gfCNCPoint4[27591] = {X 66.0153, Y 23.5146, Z -6.3333, A 0.000, B 0.000, C 0.000 }
gfCNCPoint4[27592] = {X 71.9863, Y 39.5865, Z -6.3333, A 0.000, B 0.000, C 0.000 }
gfCNCPoint4[27593] = {X 72.3293, Y 40.4492, Z -6.3333, A 0.000, B 0.000, C 0.000 }
gfCNCPoint4[27594] = {X 73.1530, Y 40.9156, Z -6.3333, A 0.000, B 0.000, C 0.000 }
gfCNCPoint4[27595] = {X 73.8471, Y 41.5593, Z -6.3333, A 0.000, B 0.000, C 0.000 }
gfCNCPoint4[27596] = {X 74.3742, Y 42.3456, Z -6.3333, A 0.000, B 0.000, C 0.000 }
gfCNCPoint4[27597] = {X 74.7059, Y 43.2322, Z -6.3333, A 0.000, B 0.000, C 0.000 }
gfCNCPoint4[27598] = {X 74.8243, Y 44.1714, Z -6.3333, A 0.000, B 0.000, C 0.000 }
gfCNCPoint4[27599] = {X 74.8245, Y 45.0000, Z -6.3333, A 0.000, B 0.000, C 0.000 }
gfCNCPoint4[27600] = {X 74.7222, Y 45.9079, Z -6.3333, A 0.000, B 0.000, C 0.000 }
gfCNCPoint4[27601] = {X 74.4204, Y 46.7702, Z -6.3333, A 0.000, B 0.000, C 0.000 }
gfCNCPoint4[27602] = {X 73.9343, Y 47.5438, Z -6.3333, A 0.000, B 0.000, C 0.000 }
gfCNCPoint4[27603] = {X 73.2883, Y 48.1899, Z -6.3333, A 0.000, B 0.000, C 0.000 }
gfCNCPoint4[27604] = {X 72.5147, Y 48.6760, Z -6.3333, A 0.000, B 0.000, C 0.000 }
gfCNCPoint4[27605] = {X 71.6523, Y 48.9777, Z -6.3333, A 0.000, B 0.000, C 0.000 }
gfCNCPoint4[27606] = {X 70.7445, Y 49.0800, Z -6.3333, A 0.000, B 0.000, C 0.000 }
gfCNCPoint4[27607] = {X 64.1851, Y 49.0800, Z -6.3333, A 0.000, B 0.000, C 0.000 }
gfCNCPoint4[27608] = {X 63.2772, Y 48.9777, Z -6.3333, A 0.000, B 0.000, C 0.000 }
gfCNCPoint4[27609] = {X 62.4149, Y 48.6760, Z -6.3333, A 0.000, B 0.000, C 0.000 }
gfCNCPoint4[27610] = {X 61.6413, Y 48.1899, Z -6.3333, A 0.000, B 0.000, C 0.000 }
gfCNCPoint4[27611] = {X 60.9953, Y 47.5438, Z -6.3333, A 0.000, B 0.000, C 0.000 }
gfCNCPoint4[27612] = {X 60.5092, Y 46.7702, Z -6.3333, A 0.000, B 0.000, C 0.000 }
gfCNCPoint4[27613] = {X 60.2074, Y 45.9079, Z -6.3333, A 0.000, B 0.000, C 0.000 }
gfCNCPoint4[27614] = {X 60.1051, Y 45.0000, Z -6.3333, A 0.000, B 0.000, C 0.000 }
gfCNCPoint4[27615] = {X 60.1051, Y 44.2086, Z -6.3333, A 0.000, B 0.000, C 0.000 }
gfCNCPoint4[27616] = {X 60.1952, Y 43.3581, Z -6.3333, A 0.000, B 0.000, C 0.000 }
gfCNCPoint4[27617] = {X 60.4606, Y 42.5451, Z -6.3333, A 0.000, B 0.000, C 0.000 }
gfCNCPoint4[27618] = {X 60.8897, Y 41.8052, Z -6.3333, A 0.000, B 0.000, C 0.000 }
gfCNCPoint4[27619] = {X 60.1744, Y 39.8492, Z -6.3333, A 0.000, B 0.000, C 0.000 }
gfCNCPoint4[27620] = {X 51.9112, Y 39.8492, Z -6.3333, A 0.000, B 0.000, C 0.000 }
gfCNCPoint4[27621] = {X 51.0699, Y 42.1094, Z -6.3333, A 0.000, B 0.000, C 0.000 }
gfCNCPoint4[27622] = {X 51.1301, Y 42.2106, Z -6.3333, A 0.000, B 0.000, C 0.000 }
gfCNCPoint4[27623] = {X 51.4138, Y 42.8326, Z -6.3333, A 0.000, B 0.000, C 0.000 }
gfCNCPoint4[27624] = {X 51.5897, Y 43.4933, Z -6.3333, A 0.000, B 0.000, C 0.000 }
gfCNCPoint4[27625] = {X 51.6528, Y 44.1740, Z -6.3333, A 0.000, B 0.000, C 0.000 }
gfCNCPoint4[27626] = {X 51.6529, Y 45.0000, Z -6.3333, A 0.000, B 0.000, C 0.000 }
gfCNCPoint4[27627] = {X 51.5506, Y 45.9079, Z -6.3333, A 0.000, B 0.000, C 0.000 }
gfCNCPoint4[27628] = {X 51.2489, Y 46.7702, Z -6.3333, A 0.000, B 0.000, C 0.000 }
gfCNCPoint4[27629] = {X 50.7628, Y 47.5438, Z -6.3333, A 0.000, B 0.000, C 0.000 }
gfCNCPoint4[27630] = {X 50.1168, Y 48.1899, Z -6.3333, A 0.000, B 0.000, C 0.000 }
gfCNCPoint4[27631] = {X 49.3432, Y 48.6760, Z -6.3333, A 0.000, B 0.000, C 0.000 }
gfCNCPoint4[27632] = {X 48.4808, Y 48.9777, Z -6.3333, A 0.000, B 0.000, C 0.000 }
gfCNCPoint4[27633] = {X 47.5729, Y 49.0800, Z -6.3333, A 0.000, B 0.000, C 0.000 }
gfCNCPoint4[27634] = {X 40.6393, Y 49.0800, Z -6.3333, A 0.000, B 0.000, C 0.000 }
gfCNCPoint4[27635] = {X 39.7314, Y 48.9777, Z -6.3333, A 0.000, B 0.000, C 0.000 }
gfCNCPoint4[27636] = {X 38.8691, Y 48.6760, Z -6.3333, A 0.000, B 0.000, C 0.000 }
gfCNCPoint4[27637] = {X 38.0955, Y 48.1899, Z -6.3333, A 0.000, B 0.000, C 0.000 }
gfCNCPoint4[27638] = {X 37.4494, Y 47.5438, Z -6.3333, A 0.000, B 0.000, C 0.000 }
gfCNCPoint4[27639] = {X 36.9633, Y 46.7702, Z -6.3333, A 0.000, B 0.000, C 0.000 }
gfCNCPoint4[27640] = {X 36.6616, Y 45.9079, Z -6.3333, A 0.000, B 0.000, C 0.000 }
gfCNCPoint4[27641] = {X 36.5593, Y 45.0000, Z -6.3333, A 0.000, B 0.000, C 0.000 }
gfCNCPoint4[27642] = {X 36.5593, Y 44.2086, Z -6.3333, A 0.000, B 0.000, C 0.000 }
gfCNCPoint4[27643] = {X 36.6734, Y 43.2505, Z -6.3333, A 0.000, B 0.000, C 0.000 }
gfCNCPoint4[27644] = {X 37.0093, Y 42.3461, Z -6.3333, A 0.000, B 0.000, C 0.000 }
gfCNCPoint4[27645] = {X 37.5482, Y 41.5458, Z -6.3333, A 0.000, B 0.000, C 0.000 }
gfCNCPoint4[27646] = {X 38.2600, Y 40.8944, Z -6.3333, A 0.000, B 0.000, C 0.000 }
gfCNCPoint4[27647] = {X 39.1048, Y 40.4284, Z -6.3333, A 0.000, B 0.000, C 0.000 }
gfCNCPoint4[27648] = {X 39.1153, Y 40.4182, Z -6.3333, A 0.000, B 0.000, C 0.000 }
gfCNCPoint4[27649] = {X 39.1252, Y 40.3961, Z -6.3333, A 0.000, B 0.000, C 0.000 }
gfCNCPoint4[27650] = {X 39.7337, Y 38.9641, Z -6.3333, A 0.000, B 0.000, C 0.000 }
gfCNCPoint4[27651] = {X 40.2895, Y 37.5107, Z -6.3333, A 0.000, B 0.000, C 0.000 }
gfCNCPoint4[27652] = {X 43.8728, Y 27.8910, Z -6.3333, A 0.000, B 0.000, C 0.000 }
gfCNCPoint4[27653] = {X 40.1244, Y 26.4948, Z -6.3333, A 0.000, B 0.000, C 0.000 }
gfCNCPoint4[27654] = {X 43.9477, Y 27.9190, Z -6.3333, A 0.000, B 0.000, C 0.000 }
gfCNCPoint4[27655] = {X 48.6479, Y 15.3010, Z -6.3333, A 0.000, B 0.000, C 0.000 }
gfCNCPoint4[27656] = {X 48.2407, Y 14.5838, Z -6.3333, A 0.000, B 0.000, C 0.000 }
gfCNCPoint4[27657] = {X 47.9892, Y 13.7983, Z -6.3333, A 0.000, B 0.000, C 0.000 }
gfCNCPoint4[27658] = {X 47.9042, Y 12.9780, Z -6.3333, A 0.000, B 0.000, C 0.000 }
gfCNCPoint4[27659] = {X 47.9042, Y 12.1868, Z -6.3333, A 0.000, B 0.000, C 0.000 }
gfCNCPoint4[27660] = {X 48.0045, Y 11.2967, Z -6.3333, A 0.000, B 0.000, C 0.000 }
gfCNCPoint4[27661] = {X 48.3003, Y 10.4513, Z -6.3333, A 0.000, B 0.000, C 0.000 }
gfCNCPoint4[27662] = {X 48.7769, Y 9.6929, Z -6.3333, A 0.000, B 0.000, C 0.000 }
gfCNCPoint4[27663] = {X 49.4103, Y 9.0595, Z -6.3333, A 0.000, B 0.000, C 0.000 }
gfCNCPoint4[27664] = {X 50.1687, Y 8.5829, Z -6.3333, A 0.000, B 0.000, C 0.000 }
gfCNCPoint4[27665] = {X 51.0141, Y 8.2871, Z -6.3333, A 0.000, B 0.000, C 0.000 }
gfCNCPoint4[27666] = {X 51.9042, Y 8.1868, Z -6.3333, A 0.000, B 0.000, C 0.000 }
gfCNCPoint4[27667] = {X 59.6221, Y 8.1868, Z -6.3333, A 0.000, B 0.000, C 0.000 }
gfCNCPoint4[27668] = {X 60.5122, Y 8.2871, Z -6.3333, A 0.000, B 0.000, C 0.000 }
gfCNCPoint4[27669] = {X 61.3577, Y 8.5829, Z -6.3333, A 0.000, B 0.000, C 0.000 }
gfCNCPoint4[27670] = {X 62.1161, Y 9.0595, Z -6.3333, A 0.000, B 0.000, C 0.000 }
gfCNCPoint4[27671] = {X 62.7495, Y 9.6929, Z -6.3333, A 0.000, B 0.000, C 0.000 }
gfCNCPoint4[27672] = {X 63.2260, Y 10.4513, Z -6.3333, A 0.000, B 0.000, C 0.000 }
gfCNCPoint4[27673] = {X 63.5218, Y 11.2967, Z -6.3333, A 0.000, B 0.000, C 0.000 }
gfCNCPoint4[27674] = {X 63.6221, Y 12.1868, Z -6.3333, A 0.000, B 0.000, C 0.000 }
gfCNCPoint4[27675] = {X 63.6219, Y 13.0192, Z -6.3333, A 0.000, B 0.000, C 0.000 }
gfCNCPoint4[27676] = {X 63.5278, Y 13.8417, Z -6.3333, A 0.000, B 0.000, C 0.000 }
gfCNCPoint4[27677] = {X 63.2663, Y 14.6272, Z -6.3333, A 0.000, B 0.000, C 0.000 }
gfCNCPoint4[27678] = {X 62.8488, Y 15.3420, Z -6.3333, A 0.000, B 0.000, C 0.000 }
gfCNCPoint4[27679] = {X 63.1271, Y 16.0764, Z -6.3333, A 0.000, B 0.000, C 0.000 }
gfCNCPoint4[27680] = {X 65.9404, Y 23.5426, Z -6.3333, A 0.000, B 0.000, C 0.000 }
gfCNCPoint4[27681] = {X 71.9117, Y 39.6152, Z -6.3333, A 0.000, B 0.000, C 0.000 }
gfCNCPoint4[27682] = {X 72.2608, Y 40.4935, Z -6.3333, A 0.000, B 0.000, C 0.000 }
gfCNCPoint4[27683] = {X 72.2699, Y 40.5075, Z -6.3333, A 0.000, B 0.000, C 0.000 }
gfCNCPoint4[27684] = {X 72.2838, Y 40.5168, Z -6.3333, A 0.000, B 0.000, C 0.000 }
gfCNCPoint4[27685] = {X 72.3479, Y 40.5442, Z -6.3333, A 0.000, B 0.000, C 0.000 }
gfCNCPoint4[27686] = {X 72.4115, Y 40.5727, Z -6.3333, A 0.000, B 0.000, C 0.000 }
gfCNCPoint4[27687] = {X 73.1908, Y 41.0441, Z -6.3333, A 0.000, B 0.000, C 0.000 }
gfCNCPoint4[27688] = {X 73.8433, Y 41.6795, Z -6.3333, A 0.000, B 0.000, C 0.000 }
gfCNCPoint4[27689] = {X 74.3351, Y 42.4461, Z -6.3333, A 0.000, B 0.000, C 0.000 }
gfCNCPoint4[27690] = {X 74.6408, Y 43.3040, Z -6.3333, A 0.000, B 0.000, C 0.000 }
gfCNCPoint4[27691] = {X 74.7445, Y 44.2089, Z -6.3333, A 0.000, B 0.000, C 0.000 }
gfCNCPoint4[27692] = {X 74.7445, Y 45.0000, Z -6.3333, A 0.000, B 0.000, C 0.000 }
gfCNCPoint4[27693] = {X 74.6442, Y 45.8901, Z -6.3333, A 0.000, B 0.000, C 0.000 }
gfCNCPoint4[27694] = {X 74.3483, Y 46.7355, Z -6.3333, A 0.000, B 0.000, C 0.000 }
gfCNCPoint4[27695] = {X 73.8718, Y 47.4940, Z -6.3333, A 0.000, B 0.000, C 0.000 }
gfCNCPoint4[27696] = {X 73.2384, Y 48.1273, Z -6.3333, A 0.000, B 0.000, C 0.000 }
gfCNCPoint4[27697] = {X 72.4800, Y 48.6039, Z -6.3333, A 0.000, B 0.000, C 0.000 }
gfCNCPoint4[27698] = {X 71.6345, Y 48.8997, Z -6.3333, A 0.000, B 0.000, C 0.000 }
gfCNCPoint4[27699] = {X 70.7445, Y 49.0000, Z -6.3333, A 0.000, B 0.000, C 0.000 }
gfCNCPoint4[27700] = {X 64.1851, Y 49.0000, Z -6.3333, A 0.000, B 0.000, C 0.000 }
gfCNCPoint4[27701] = {X 63.2951, Y 48.8997, Z -6.3333, A 0.000, B 0.000, C 0.000 }
gfCNCPoint4[27702] = {X 62.4496, Y 48.6039, Z -6.3333, A 0.000, B 0.000, C 0.000 }
gfCNCPoint4[27703] = {X 61.6912, Y 48.1273, Z -6.3333, A 0.000, B 0.000, C 0.000 }
gfCNCPoint4[27704] = {X 61.0578, Y 47.4940, Z -6.3333, A 0.000, B 0.000, C 0.000 }
gfCNCPoint4[27705] = {X 60.5813, Y 46.7355, Z -6.3333, A 0.000, B 0.000, C 0.000 }
gfCNCPoint4[27706] = {X 60.2854, Y 45.8901, Z -6.3333, A 0.000, B 0.000, C 0.000 }
gfCNCPoint4[27707] = {X 60.1851, Y 45.0000, Z -6.3333, A 0.000, B 0.000, C 0.000 }
gfCNCPoint4[27708] = {X 60.1855, Y 44.1538, Z -6.3333, A 0.000, B 0.000, C 0.000 }
gfCNCPoint4[27709] = {X 60.2746, Y 43.3674, Z -6.3333, A 0.000, B 0.000, C 0.000 }
gfCNCPoint4[27710] = {X 60.5168, Y 42.6140, Z -6.3333, A 0.000, B 0.000, C 0.000 }
gfCNCPoint4[27711] = {X 60.9025, Y 41.9231, Z -6.3333, A 0.000, B 0.000, C 0.000 }
gfCNCPoint4[27712] = {X 60.9795, Y 41.8179, Z -6.3333, A 0.000, B 0.000, C 0.000 }
gfCNCPoint4[27713] = {X 60.2304, Y 39.7692, Z -6.3333, A 0.000, B 0.000, C 0.000 }
gfCNCPoint4[27714] = {X 51.8428, Y 39.7692, Z -6.3333, A 0.000, B 0.000, C 0.000 }
gfCNCPoint4[27715] = {X 51.8428, Y 39.8035, Z -6.3333, A 0.000, B 0.000, C 0.000 }
gfCNCPoint4[27716] = {X 50.9816, Y 42.1174, Z -6.3333, A 0.000, B 0.000, C 0.000 }
gfCNCPoint4[27717] = {X 51.0729, Y 42.2722, Z -6.3333, A 0.000, B 0.000, C 0.000 }
gfCNCPoint4[27718] = {X 51.3480, Y 42.8865, Z -6.3333, A 0.000, B 0.000, C 0.000 }
gfCNCPoint4[27719] = {X 51.5163, Y 43.5382, Z -6.3333, A 0.000, B 0.000, C 0.000 }
gfCNCPoint4[27720] = {X 51.5729, Y 44.2089, Z -6.3333, A 0.000, B 0.000, C 0.000 }
gfCNCPoint4[27721] = {X 51.5729, Y 45.0000, Z -6.3333, A 0.000, B 0.000, C 0.000 }
gfCNCPoint4[27722] = {X 51.4726, Y 45.8901, Z -6.3333, A 0.000, B 0.000, C 0.000 }
gfCNCPoint4[27723] = {X 51.1768, Y 46.7355, Z -6.3333, A 0.000, B 0.000, C 0.000 }
gfCNCPoint4[27724] = {X 50.7003, Y 47.4940, Z -6.3333, A 0.000, B 0.000, C 0.000 }
gfCNCPoint4[27725] = {X 50.0669, Y 48.1273, Z -6.3333, A 0.000, B 0.000, C 0.000 }
gfCNCPoint4[27726] = {X 49.3085, Y 48.6039, Z -6.3333, A 0.000, B 0.000, C 0.000 }
gfCNCPoint4[27727] = {X 48.4630, Y 48.8997, Z -6.3333, A 0.000, B 0.000, C 0.000 }
gfCNCPoint4[27728] = {X 47.5729, Y 49.0000, Z -6.3333, A 0.000, B 0.000, C 0.000 }
gfCNCPoint4[27729] = {X 40.6393, Y 49.0000, Z -6.3333, A 0.000, B 0.000, C 0.000 }
gfCNCPoint4[27730] = {X 39.7492, Y 48.8997, Z -6.3333, A 0.000, B 0.000, C 0.000 }
gfCNCPoint4[27731] = {X 38.9038, Y 48.6039, Z -6.3333, A 0.000, B 0.000, C 0.000 }
gfCNCPoint4[27732] = {X 38.1453, Y 48.1273, Z -6.3333, A 0.000, B 0.000, C 0.000 }
gfCNCPoint4[27733] = {X 37.5120, Y 47.4940, Z -6.3333, A 0.000, B 0.000, C 0.000 }
gfCNCPoint4[27734] = {X 37.0354, Y 46.7355, Z -6.3333, A 0.000, B 0.000, C 0.000 }
gfCNCPoint4[27735] = {X 36.7396, Y 45.8901, Z -6.3333, A 0.000, B 0.000, C 0.000 }
gfCNCPoint4[27736] = {X 36.6393, Y 45.0000, Z -6.3333, A 0.000, B 0.000, C 0.000 }
gfCNCPoint4[27737] = {X 36.6397, Y 44.1538, Z -6.3333, A 0.000, B 0.000, C 0.000 }
gfCNCPoint4[27738] = {X 36.7563, Y 43.2484, Z -6.3333, A 0.000, B 0.000, C 0.000 }
gfCNCPoint4[27739] = {X 37.0752, Y 42.3931, Z -6.3333, A 0.000, B 0.000, C 0.000 }
gfCNCPoint4[27740] = {X 37.5796, Y 41.6323, Z -6.3333, A 0.000, B 0.000, C 0.000 }
gfCNCPoint4[27741] = {X 38.2434, Y 41.0057, Z -6.3333, A 0.000, B 0.000, C 0.000 }
gfCNCPoint4[27742] = {X 39.0320, Y 40.5459, Z -6.3333, A 0.000, B 0.000, C 0.000 }
gfCNCPoint4[27743] = {X 39.0833, Y 40.5238, Z -6.3333, A 0.000, B 0.000, C 0.000 }
gfCNCPoint4[27744] = {X 39.1349, Y 40.5025, Z -6.3333, A 0.000, B 0.000, C 0.000 }
gfCNCPoint4[27745] = {X 39.1666, Y 40.4818, Z -6.3333, A 0.000, B 0.000, C 0.000 }
gfCNCPoint4[27746] = {X 39.1883, Y 40.4509, Z -6.3333, A 0.000, B 0.000, C 0.000 }
gfCNCPoint4[27747] = {X 39.2126, Y 40.3964, Z -6.3333, A 0.000, B 0.000, C 0.000 }
gfCNCPoint4[27748] = {X 39.2369, Y 40.3420, Z -6.3333, A 0.000, B 0.000, C 0.000 }
gfCNCPoint4[27749] = {X 39.8256, Y 38.9501, Z -6.3333, A 0.000, B 0.000, C 0.000 }
gfCNCPoint4[27750] = {X 40.3646, Y 37.5383, Z -6.3333, A 0.000, B 0.000, C 0.000 }
gfCNCPoint4[27751] = {X 43.9477, Y 27.9190, Z -6.3333, A 0.000, B 0.000, C 0.000 }
gfCNCPoint4[27752] = {X 40.1244, Y 26.4948, Z -6.3333, A 0.000, B 0.000, C 0.000 }
gfCNCPoint4[27753] = {X 40.1244, Y 26.4948, Z -3.3333, A 0.000, B 0.000, C 0.000 }
gfCNCPoint4[27754] = {X 40.1244, Y 26.4948, Z 11.0000, A 0.000, B 0.000, C 0.000 }
gfCNCPoint4[27755] = {X 79.0220, Y 28.5912, Z 11.0000, A 0.000, B 0.000, C 0.000 }
gfCNCPoint4[27756] = {X 79.0220, Y 28.5912, Z -3.3333, A 0.000, B 0.000, C 0.000 }
gfCNCPoint4[27757] = {X 79.0220, Y 28.5912, Z -6.3333, A 0.000, B 0.000, C 0.000 }
gfCNCPoint4[27758] = {X 83.1020, Y 28.5912, Z -6.3333, A 0.000, B 0.000, C 0.000 }
gfCNCPoint4[27759] = {X 83.1019, Y 16.2736, Z -6.3333, A 0.000, B 0.000, C 0.000 }
gfCNCPoint4[27760] = {X 82.4637, Y 15.6025, Z -6.3333, A 0.000, B 0.000, C 0.000 }
gfCNCPoint4[27761] = {X 81.9831, Y 14.8108, Z -6.3333, A 0.000, B 0.000, C 0.000 }
gfCNCPoint4[27762] = {X 81.6824, Y 13.9349, Z -6.3333, A 0.000, B 0.000, C 0.000 }
gfCNCPoint4[27763] = {X 81.5752, Y 13.0150, Z -6.3333, A 0.000, B 0.000, C 0.000 }
gfCNCPoint4[27764] = {X 81.5751, Y 12.1868, Z -6.3333, A 0.000, B 0.000, C 0.000 }
gfCNCPoint4[27765] = {X 81.6834, Y 11.2255, Z -6.3333, A 0.000, B 0.000, C 0.000 }
gfCNCPoint4[27766] = {X 82.0029, Y 10.3125, Z -6.3333, A 0.000, B 0.000, C 0.000 }
gfCNCPoint4[27767] = {X 82.5176, Y 9.4933, Z -6.3333, A 0.000, B 0.000, C 0.000 }
gfCNCPoint4[27768] = {X 83.2016, Y 8.8093, Z -6.3333, A 0.000, B 0.000, C 0.000 }
gfCNCPoint4[27769] = {X 84.0207, Y 8.2946, Z -6.3333, A 0.000, B 0.000, C 0.000 }
gfCNCPoint4[27770] = {X 84.9338, Y 7.9751, Z -6.3333, A 0.000, B 0.000, C 0.000 }
gfCNCPoint4[27771] = {X 85.8951, Y 7.8668, Z -6.3333, A 0.000, B 0.000, C 0.000 }
gfCNCPoint4[27772] = {X 94.0497, Y 7.8668, Z -6.3333, A 0.000, B 0.000, C 0.000 }
gfCNCPoint4[27773] = {X 95.0110, Y 7.9751, Z -6.3333, A 0.000, B 0.000, C 0.000 }
gfCNCPoint4[27774] = {X 95.9240, Y 8.2946, Z -6.3333, A 0.000, B 0.000, C 0.000 }
gfCNCPoint4[27775] = {X 96.7431, Y 8.8093, Z -6.3333, A 0.000, B 0.000, C 0.000 }
gfCNCPoint4[27776] = {X 97.4272, Y 9.4933, Z -6.3333, A 0.000, B 0.000, C 0.000 }
gfCNCPoint4[27777] = {X 97.9419, Y 10.3124, Z -6.3333, A 0.000, B 0.000, C 0.000 }
gfCNCPoint4[27778] = {X 98.2614, Y 11.2255, Z -6.3333, A 0.000, B 0.000, C 0.000 }
gfCNCPoint4[27779] = {X 98.3697, Y 12.1868, Z -6.3333, A 0.000, B 0.000, C 0.000 }
gfCNCPoint4[27780] = {X 98.3697, Y 12.9782, Z -6.3333, A 0.000, B 0.000, C 0.000 }
gfCNCPoint4[27781] = {X 98.2967, Y 13.7678, Z -6.3333, A 0.000, B 0.000, C 0.000 }
gfCNCPoint4[27782] = {X 98.0807, Y 14.5307, Z -6.3333, A 0.000, B 0.000, C 0.000 }
gfCNCPoint4[27783] = {X 97.7289, Y 15.2414, Z -6.3333, A 0.000, B 0.000, C 0.000 }
gfCNCPoint4[27784] = {X 101.8758, Y 25.5228, Z -6.3333, A 0.000, B 0.000, C 0.000 }
gfCNCPoint4[27785] = {X 106.0162, Y 15.2210, Z -6.3333, A 0.000, B 0.000, C 0.000 }
gfCNCPoint4[27786] = {X 105.6760, Y 14.5282, Z -6.3333, A 0.000, B 0.000, C 0.000 }
gfCNCPoint4[27787] = {X 105.4645, Y 13.7860, Z -6.3333, A 0.000, B 0.000, C 0.000 }
gfCNCPoint4[27788] = {X 105.3885, Y 13.0179, Z -6.3333, A 0.000, B 0.000, C 0.000 }
gfCNCPoint4[27789] = {X 105.3883, Y 12.1868, Z -6.3333, A 0.000, B 0.000, C 0.000 }
gfCNCPoint4[27790] = {X 105.4966, Y 11.2255, Z -6.3333, A 0.000, B 0.000, C 0.000 }
gfCNCPoint4[27791] = {X 105.8161, Y 10.3124, Z -6.3333, A 0.000, B 0.000, C 0.000 }
gfCNCPoint4[27792] = {X 106.3308, Y 9.4933, Z -6.3333, A 0.000, B 0.000, C 0.000 }
gfCNCPoint4[27793] = {X 107.0148, Y 8.8093, Z -6.3333, A 0.000, B 0.000, C 0.000 }
gfCNCPoint4[27794] = {X 107.8339, Y 8.2946, Z -6.3333, A 0.000, B 0.000, C 0.000 }
gfCNCPoint4[27795] = {X 108.7470, Y 7.9751, Z -6.3333, A 0.000, B 0.000, C 0.000 }
gfCNCPoint4[27796] = {X 109.7083, Y 7.8668, Z -6.3333, A 0.000, B 0.000, C 0.000 }
gfCNCPoint4[27797] = {X 117.7916, Y 7.8668, Z -6.3333, A 0.000, B 0.000, C 0.000 }
gfCNCPoint4[27798] = {X 118.7529, Y 7.9751, Z -6.3333, A 0.000, B 0.000, C 0.000 }
gfCNCPoint4[27799] = {X 119.6660, Y 8.2946, Z -6.3333, A 0.000, B 0.000, C 0.000 }
gfCNCPoint4[27800] = {X 120.4851, Y 8.8093, Z -6.3333, A 0.000, B 0.000, C 0.000 }
gfCNCPoint4[27801] = {X 121.1691, Y 9.4933, Z -6.3333, A 0.000, B 0.000, C 0.000 }
gfCNCPoint4[27802] = {X 121.6838, Y 10.3124, Z -6.3333, A 0.000, B 0.000, C 0.000 }
gfCNCPoint4[27803] = {X 122.0033, Y 11.2255, Z -6.3333, A 0.000, B 0.000, C 0.000 }
gfCNCPoint4[27804] = {X 122.1116, Y 12.1868, Z -6.3333, A 0.000, B 0.000, C 0.000 }
gfCNCPoint4[27805] = {X 122.1116, Y 12.9782, Z -6.3333, A 0.000, B 0.000, C 0.000 }
gfCNCPoint4[27806] = {X 122.0103, Y 13.9078, Z -6.3333, A 0.000, B 0.000, C 0.000 }
gfCNCPoint4[27807] = {X 121.7114, Y 14.7939, Z -6.3333, A 0.000, B 0.000, C 0.000 }
gfCNCPoint4[27808] = {X 121.2288, Y 15.5949, Z -6.3333, A 0.000, B 0.000, C 0.000 }
gfCNCPoint4[27809] = {X 120.5851, Y 16.2732, Z -6.3333, A 0.000, B 0.000, C 0.000 }
gfCNCPoint4[27810] = {X 120.5847, Y 40.9145, Z -6.3333, A 0.000, B 0.000, C 0.000 }
gfCNCPoint4[27811] = {X 120.6226, Y 40.9457, Z -6.3333, A 0.000, B 0.000, C 0.000 }
gfCNCPoint4[27812] = {X 121.2458, Y 41.6145, Z -6.3333, A 0.000, B 0.000, C 0.000 }
gfCNCPoint4[27813] = {X 121.7144, Y 42.3993, Z -6.3333, A 0.000, B 0.000, C 0.000 }
gfCNCPoint4[27814] = {X 122.0073, Y 43.2652, Z -6.3333, A 0.000, B 0.000, C 0.000 }
gfCNCPoint4[27815] = {X 122.1114, Y 44.1734, Z -6.3333, A 0.000, B 0.000, C 0.000 }
gfCNCPoint4[27816] = {X 122.1116, Y 45.0000, Z -6.3333, A 0.000, B 0.000, C 0.000 }
gfCNCPoint4[27817] = {X 122.0033, Y 45.9613, Z -6.3333, A 0.000, B 0.000, C 0.000 }
gfCNCPoint4[27818] = {X 121.6838, Y 46.8744, Z -6.3333, A 0.000, B 0.000, C 0.000 }
gfCNCPoint4[27819] = {X 121.1691, Y 47.6935, Z -6.3333, A 0.000, B 0.000, C 0.000 }
gfCNCPoint4[27820] = {X 120.4851, Y 48.3775, Z -6.3333, A 0.000, B 0.000, C 0.000 }
gfCNCPoint4[27821] = {X 119.6660, Y 48.8922, Z -6.3333, A 0.000, B 0.000, C 0.000 }
gfCNCPoint4[27822] = {X 118.7529, Y 49.2117, Z -6.3333, A 0.000, B 0.000, C 0.000 }
gfCNCPoint4[27823] = {X 117.7916, Y 49.3200, Z -6.3333, A 0.000, B 0.000, C 0.000 }
gfCNCPoint4[27824] = {X 111.9185, Y 49.3200, Z -6.3333, A 0.000, B 0.000, C 0.000 }
gfCNCPoint4[27825] = {X 110.9619, Y 49.2128, Z -6.3333, A 0.000, B 0.000, C 0.000 }
gfCNCPoint4[27826] = {X 110.0529, Y 48.8964, Z -6.3333, A 0.000, B 0.000, C 0.000 }
gfCNCPoint4[27827] = {X 109.2365, Y 48.3866, Z -6.3333, A 0.000, B 0.000, C 0.000 }
gfCNCPoint4[27828] = {X 108.5532, Y 47.7087, Z -6.3333, A 0.000, B 0.000, C 0.000 }
gfCNCPoint4[27829] = {X 108.0369, Y 46.8963, Z -6.3333, A 0.000, B 0.000, C 0.000 }
gfCNCPoint4[27830] = {X 107.7134, Y 45.9898, Z -6.3333, A 0.000, B 0.000, C 0.000 }
gfCNCPoint4[27831] = {X 107.5986, Y 45.0341, Z -6.3333, A 0.000, B 0.000, C 0.000 }
gfCNCPoint4[27832] = {X 107.5985, Y 44.1789, Z -6.3333, A 0.000, B 0.000, C 0.000 }
gfCNCPoint4[27833] = {X 107.6340, Y 43.6366, Z -6.3333, A 0.000, B 0.000, C 0.000 }
gfCNCPoint4[27834] = {X 107.7400, Y 43.1035, Z -6.3333, A 0.000, B 0.000, C 0.000 }
gfCNCPoint4[27835] = {X 107.9081, Y 42.6047, Z -6.3333, A 0.000, B 0.000, C 0.000 }
gfCNCPoint4[27836] = {X 108.1379, Y 42.1311, Z -6.3333, A 0.000, B 0.000, C 0.000 }
gfCNCPoint4[27837] = {X 108.5875, Y 41.4624, Z -6.3333, A 0.000, B 0.000, C 0.000 }
gfCNCPoint4[27838] = {X 109.1253, Y 40.8623, Z -6.3333, A 0.000, B 0.000, C 0.000 }
gfCNCPoint4[27839] = {X 109.1252, Y 39.2978, Z -6.3333, A 0.000, B 0.000, C 0.000 }
gfCNCPoint4[27840] = {X 106.1118, Y 46.6615, Z -6.3333, A 0.000, B 0.000, C 0.000 }
gfCNCPoint4[27841] = {X 105.7417, Y 47.3611, Z -6.3333, A 0.000, B 0.000, C 0.000 }
gfCNCPoint4[27842] = {X 105.2502, Y 47.9815, Z -6.3333, A 0.000, B 0.000, C 0.000 }
gfCNCPoint4[27843] = {X 104.6538, Y 48.5018, Z -6.3333, A 0.000, B 0.000, C 0.000 }
gfCNCPoint4[27844] = {X 103.9724, Y 48.9046, Z -6.3333, A 0.000, B 0.000, C 0.000 }
gfCNCPoint4[27845] = {X 103.0287, Y 49.2242, Z -6.3333, A 0.000, B 0.000, C 0.000 }
gfCNCPoint4[27846] = {X 102.0368, Y 49.3191, Z -6.3333, A 0.000, B 0.000, C 0.000 }
gfCNCPoint4[27847] = {X 101.0496, Y 49.1842, Z -6.3333, A 0.000, B 0.000, C 0.000 }
gfCNCPoint4[27848] = {X 100.1195, Y 48.8268, Z -6.3333, A 0.000, B 0.000, C 0.000 }
gfCNCPoint4[27849] = {X 99.2961, Y 48.2657, Z -6.3333, A 0.000, B 0.000, C 0.000 }
gfCNCPoint4[27850] = {X 98.6231, Y 47.5309, Z -6.3333, A 0.000, B 0.000, C 0.000 }
gfCNCPoint4[27851] = {X 98.1363, Y 46.6615, Z -6.3333, A 0.000, B 0.000, C 0.000 }
gfCNCPoint4[27852] = {X 95.1317, Y 39.3133, Z -6.3333, A 0.000, B 0.000, C 0.000 }
gfCNCPoint4[27853] = {X 95.1317, Y 40.9048, Z -6.3333, A 0.000, B 0.000, C 0.000 }
gfCNCPoint4[27854] = {X 95.6575, Y 41.4431, Z -6.3333, A 0.000, B 0.000, C 0.000 }
gfCNCPoint4[27855] = {X 96.0839, Y 42.0632, Z -6.3333, A 0.000, B 0.000, C 0.000 }
gfCNCPoint4[27856] = {X 96.3313, Y 42.5720, Z -6.3333, A 0.000, B 0.000, C 0.000 }
gfCNCPoint4[27857] = {X 96.5113, Y 43.1084, Z -6.3333, A 0.000, B 0.000, C 0.000 }
gfCNCPoint4[27858] = {X 96.6196, Y 43.6529, Z -6.3333, A 0.000, B 0.000, C 0.000 }
gfCNCPoint4[27859] = {X 96.6585, Y 44.2066, Z -6.3333, A 0.000, B 0.000, C 0.000 }
gfCNCPoint4[27860] = {X 96.6583, Y 45.0415, Z -6.3333, A 0.000, B 0.000, C 0.000 }
gfCNCPoint4[27861] = {X 96.5422, Y 45.9960, Z -6.3333, A 0.000, B 0.000, C 0.000 }
gfCNCPoint4[27862] = {X 96.2178, Y 46.9011, Z -6.3333, A 0.000, B 0.000, C 0.000 }
gfCNCPoint4[27863] = {X 95.7012, Y 47.7120, Z -6.3333, A 0.000, B 0.000, C 0.000 }
gfCNCPoint4[27864] = {X 95.0181, Y 48.3886, Z -6.3333, A 0.000, B 0.000, C 0.000 }
gfCNCPoint4[27865] = {X 94.2022, Y 48.8973, Z -6.3333, A 0.000, B 0.000, C 0.000 }
gfCNCPoint4[27866] = {X 93.2940, Y 49.2130, Z -6.3333, A 0.000, B 0.000, C 0.000 }
gfCNCPoint4[27867] = {X 92.3385, Y 49.3200, Z -6.3333, A 0.000, B 0.000, C 0.000 }
gfCNCPoint4[27868] = {X 85.8951, Y 49.3200, Z -6.3333, A 0.000, B 0.000, C 0.000 }
gfCNCPoint4[27869] = {X 84.9387, Y 49.2128, Z -6.3333, A 0.000, B 0.000, C 0.000 }
gfCNCPoint4[27870] = {X 84.0297, Y 48.8965, Z -6.3333, A 0.000, B 0.000, C 0.000 }
gfCNCPoint4[27871] = {X 83.2134, Y 48.3869, Z -6.3333, A 0.000, B 0.000, C 0.000 }
gfCNCPoint4[27872] = {X 82.5301, Y 47.7091, Z -6.3333, A 0.000, B 0.000, C 0.000 }
gfCNCPoint4[27873] = {X 82.0138, Y 46.8970, Z -6.3333, A 0.000, B 0.000, C 0.000 }
gfCNCPoint4[27874] = {X 81.6902, Y 45.9906, Z -6.3333, A 0.000, B 0.000, C 0.000 }
gfCNCPoint4[27875] = {X 81.5752, Y 45.0351, Z -6.3333, A 0.000, B 0.000, C 0.000 }
gfCNCPoint4[27876] = {X 81.5751, Y 44.2072, Z -6.3333, A 0.000, B 0.000, C 0.000 }
gfCNCPoint4[27877] = {X 81.6799, Y 43.2778, Z -6.3333, A 0.000, B 0.000, C 0.000 }
gfCNCPoint4[27878] = {X 81.9799, Y 42.3919, Z -6.3333, A 0.000, B 0.000, C 0.000 }
gfCNCPoint4[27879] = {X 82.4613, Y 41.5900, Z -6.3333, A 0.000, B 0.000, C 0.000 }
gfCNCPoint4[27880] = {X 83.1022, Y 40.9088, Z -6.3333, A 0.000, B 0.000, C 0.000 }
gfCNCPoint4[27881] = {X 83.1020, Y 28.5912, Z -6.3333, A 0.000, B 0.000, C 0.000 }
gfCNCPoint4[27882] = {X 79.1020, Y 28.5912, Z -6.3333, A 0.000, B 0.000, C 0.000 }
gfCNCPoint4[27883] = {X 83.1820, Y 28.5912, Z -6.3333, A 0.000, B 0.000, C 0.000 }
gfCNCPoint4[27884] = {X 83.1819, Y 16.2363, Z -6.3333, A 0.000, B 0.000, C 0.000 }
gfCNCPoint4[27885] = {X 82.5441, Y 15.5758, Z -6.3333, A 0.000, B 0.000, C 0.000 }
gfCNCPoint4[27886] = {X 82.0634, Y 14.7936, Z -6.3333, A 0.000, B 0.000, C 0.000 }
gfCNCPoint4[27887] = {X 81.7624, Y 13.9262, Z -6.3333, A 0.000, B 0.000, C 0.000 }
gfCNCPoint4[27888] = {X 81.6552, Y 13.0143, Z -6.3333, A 0.000, B 0.000, C 0.000 }
gfCNCPoint4[27889] = {X 81.6551, Y 12.1868, Z -6.3333, A 0.000, B 0.000, C 0.000 }
gfCNCPoint4[27890] = {X 81.7614, Y 11.2433, Z -6.3333, A 0.000, B 0.000, C 0.000 }
gfCNCPoint4[27891] = {X 82.0750, Y 10.3472, Z -6.3333, A 0.000, B 0.000, C 0.000 }
gfCNCPoint4[27892] = {X 82.5801, Y 9.5432, Z -6.3333, A 0.000, B 0.000, C 0.000 }
gfCNCPoint4[27893] = {X 83.2515, Y 8.8719, Z -6.3333, A 0.000, B 0.000, C 0.000 }
gfCNCPoint4[27894] = {X 84.0554, Y 8.3667, Z -6.3333, A 0.000, B 0.000, C 0.000 }
gfCNCPoint4[27895] = {X 84.9516, Y 8.0531, Z -6.3333, A 0.000, B 0.000, C 0.000 }
gfCNCPoint4[27896] = {X 85.8951, Y 7.9468, Z -6.3333, A 0.000, B 0.000, C 0.000 }
gfCNCPoint4[27897] = {X 94.0497, Y 7.9468, Z -6.3333, A 0.000, B 0.000, C 0.000 }
gfCNCPoint4[27898] = {X 94.9932, Y 8.0531, Z -6.3333, A 0.000, B 0.000, C 0.000 }
gfCNCPoint4[27899] = {X 95.8893, Y 8.3667, Z -6.3333, A 0.000, B 0.000, C 0.000 }
gfCNCPoint4[27900] = {X 96.6933, Y 8.8718, Z -6.3333, A 0.000, B 0.000, C 0.000 }
gfCNCPoint4[27901] = {X 97.3646, Y 9.5432, Z -6.3333, A 0.000, B 0.000, C 0.000 }
gfCNCPoint4[27902] = {X 97.8698, Y 10.3471, Z -6.3333, A 0.000, B 0.000, C 0.000 }
gfCNCPoint4[27903] = {X 98.1834, Y 11.2433, Z -6.3333, A 0.000, B 0.000, C 0.000 }
gfCNCPoint4[27904] = {X 98.2897, Y 12.1868, Z -6.3333, A 0.000, B 0.000, C 0.000 }
gfCNCPoint4[27905] = {X 98.2897, Y 12.9782, Z -6.3333, A 0.000, B 0.000, C 0.000 }
gfCNCPoint4[27906] = {X 98.2156, Y 13.7663, Z -6.3333, A 0.000, B 0.000, C 0.000 }
gfCNCPoint4[27907] = {X 97.9963, Y 14.5270, Z -6.3333, A 0.000, B 0.000, C 0.000 }
gfCNCPoint4[27908] = {X 97.6395, Y 15.2336, Z -6.3333, A 0.000, B 0.000, C 0.000 }
gfCNCPoint4[27909] = {X 101.8760, Y 25.7370, Z -6.3333, A 0.000, B 0.000, C 0.000 }
gfCNCPoint4[27910] = {X 106.1054, Y 15.2135, Z -6.3333, A 0.000, B 0.000, C 0.000 }
gfCNCPoint4[27911] = {X 105.7603, Y 14.5243, Z -6.3333, A 0.000, B 0.000, C 0.000 }
gfCNCPoint4[27912] = {X 105.5456, Y 13.7841, Z -6.3333, A 0.000, B 0.000, C 0.000 }
gfCNCPoint4[27913] = {X 105.4685, Y 13.0172, Z -6.3333, A 0.000, B 0.000, C 0.000 }
gfCNCPoint4[27914] = {X 105.4683, Y 12.1868, Z -6.3333, A 0.000, B 0.000, C 0.000 }
gfCNCPoint4[27915] = {X 105.5746, Y 11.2433, Z -6.3333, A 0.000, B 0.000, C 0.000 }
gfCNCPoint4[27916] = {X 105.8882, Y 10.3471, Z -6.3333, A 0.000, B 0.000, C 0.000 }
gfCNCPoint4[27917] = {X 106.3933, Y 9.5432, Z -6.3333, A 0.000, B 0.000, C 0.000 }
gfCNCPoint4[27918] = {X 107.0647, Y 8.8718, Z -6.3333, A 0.000, B 0.000, C 0.000 }
gfCNCPoint4[27919] = {X 107.8686, Y 8.3667, Z -6.3333, A 0.000, B 0.000, C 0.000 }
gfCNCPoint4[27920] = {X 108.7648, Y 8.0531, Z -6.3333, A 0.000, B 0.000, C 0.000 }
gfCNCPoint4[27921] = {X 109.7083, Y 7.9468, Z -6.3333, A 0.000, B 0.000, C 0.000 }
gfCNCPoint4[27922] = {X 117.7916, Y 7.9468, Z -6.3333, A 0.000, B 0.000, C 0.000 }
gfCNCPoint4[27923] = {X 118.7351, Y 8.0531, Z -6.3333, A 0.000, B 0.000, C 0.000 }
gfCNCPoint4[27924] = {X 119.6312, Y 8.3667, Z -6.3333, A 0.000, B 0.000, C 0.000 }
gfCNCPoint4[27925] = {X 120.4352, Y 8.8718, Z -6.3333, A 0.000, B 0.000, C 0.000 }
gfCNCPoint4[27926] = {X 121.1065, Y 9.5432, Z -6.3333, A 0.000, B 0.000, C 0.000 }
gfCNCPoint4[27927] = {X 121.6117, Y 10.3471, Z -6.3333, A 0.000, B 0.000, C 0.000 }
gfCNCPoint4[27928] = {X 121.9253, Y 11.2433, Z -6.3333, A 0.000, B 0.000, C 0.000 }
gfCNCPoint4[27929] = {X 122.0316, Y 12.1868, Z -6.3333, A 0.000, B 0.000, C 0.000 }
gfCNCPoint4[27930] = {X 122.0316, Y 12.9782, Z -6.3333, A 0.000, B 0.000, C 0.000 }
gfCNCPoint4[27931] = {X 121.9302, Y 13.8996, Z -6.3333, A 0.000, B 0.000, C 0.000 }
gfCNCPoint4[27932] = {X 121.6310, Y 14.7770, Z -6.3333, A 0.000, B 0.000, C 0.000 }
gfCNCPoint4[27933] = {X 121.1483, Y 15.5684, Z -6.3333, A 0.000, B 0.000, C 0.000 }
gfCNCPoint4[27934] = {X 120.5051, Y 16.2360, Z -6.3333, A 0.000, B 0.000, C 0.000 }
gfCNCPoint4[27935] = {X 120.5047, Y 40.9523, Z -6.3333, A 0.000, B 0.000, C 0.000 }
gfCNCPoint4[27936] = {X 120.5710, Y 41.0068, Z -6.3333, A 0.000, B 0.000, C 0.000 }
gfCNCPoint4[27937] = {X 121.1823, Y 41.6631, Z -6.3333, A 0.000, B 0.000, C 0.000 }
gfCNCPoint4[27938] = {X 121.6419, Y 42.4333, Z -6.3333, A 0.000, B 0.000, C 0.000 }
gfCNCPoint4[27939] = {X 121.9293, Y 43.2830, Z -6.3333, A 0.000, B 0.000, C 0.000 }
gfCNCPoint4[27940] = {X 122.0314, Y 44.1740, Z -6.3333, A 0.000, B 0.000, C 0.000 }
gfCNCPoint4[27941] = {X 122.0316, Y 45.0000, Z -6.3333, A 0.000, B 0.000, C 0.000 }
gfCNCPoint4[27942] = {X 121.9253, Y 45.9435, Z -6.3333, A 0.000, B 0.000, C 0.000 }
gfCNCPoint4[27943] = {X 121.6117, Y 46.8397, Z -6.3333, A 0.000, B 0.000, C 0.000 }
gfCNCPoint4[27944] = {X 121.1065, Y 47.6436, Z -6.3333, A 0.000, B 0.000, C 0.000 }
gfCNCPoint4[27945] = {X 120.4352, Y 48.3150, Z -6.3333, A 0.000, B 0.000, C 0.000 }
gfCNCPoint4[27946] = {X 119.6312, Y 48.8201, Z -6.3333, A 0.000, B 0.000, C 0.000 }
gfCNCPoint4[27947] = {X 118.7351, Y 49.1337, Z -6.3333, A 0.000, B 0.000, C 0.000 }
gfCNCPoint4[27948] = {X 117.7916, Y 49.2400, Z -6.3333, A 0.000, B 0.000, C 0.000 }
gfCNCPoint4[27949] = {X 111.9185, Y 49.2400, Z -6.3333, A 0.000, B 0.000, C 0.000 }
gfCNCPoint4[27950] = {X 110.9797, Y 49.1348, Z -6.3333, A 0.000, B 0.000, C 0.000 }
gfCNCPoint4[27951] = {X 110.0874, Y 48.8242, Z -6.3333, A 0.000, B 0.000, C 0.000 }
gfCNCPoint4[27952] = {X 109.2861, Y 48.3239, Z -6.3333, A 0.000, B 0.000, C 0.000 }
gfCNCPoint4[27953] = {X 108.6155, Y 47.6585, Z -6.3333, A 0.000, B 0.000, C 0.000 }
gfCNCPoint4[27954] = {X 108.1088, Y 46.8612, Z -6.3333, A 0.000, B 0.000, C 0.000 }
gfCNCPoint4[27955] = {X 107.7913, Y 45.9714, Z -6.3333, A 0.000, B 0.000, C 0.000 }
gfCNCPoint4[27956] = {X 107.6786, Y 45.0335, Z -6.3333, A 0.000, B 0.000, C 0.000 }
gfCNCPoint4[27957] = {X 107.6785, Y 44.1789, Z -6.3333, A 0.000, B 0.000, C 0.000 }
gfCNCPoint4[27958] = {X 107.7133, Y 43.6470, Z -6.3333, A 0.000, B 0.000, C 0.000 }
gfCNCPoint4[27959] = {X 107.8173, Y 43.1242, Z -6.3333, A 0.000, B 0.000, C 0.000 }
gfCNCPoint4[27960] = {X 107.9822, Y 42.6350, Z -6.3333, A 0.000, B 0.000, C 0.000 }
gfCNCPoint4[27961] = {X 108.2075, Y 42.1705, Z -6.3333, A 0.000, B 0.000, C 0.000 }
gfCNCPoint4[27962] = {X 108.6612, Y 41.4980, Z -6.3333, A 0.000, B 0.000, C 0.000 }
gfCNCPoint4[27963] = {X 109.2053, Y 40.8963, Z -6.3333, A 0.000, B 0.000, C 0.000 }
gfCNCPoint4[27964] = {X 109.2051, Y 39.1629, Z -6.3333, A 0.000, B 0.000, C 0.000 }
gfCNCPoint4[27965] = {X 109.0939, Y 39.1629, Z -6.3333, A 0.000, B 0.000, C 0.000 }
gfCNCPoint4[27966] = {X 106.0379, Y 46.6307, Z -6.3333, A 0.000, B 0.000, C 0.000 }
gfCNCPoint4[27967] = {X 105.6747, Y 47.3174, Z -6.3333, A 0.000, B 0.000, C 0.000 }
gfCNCPoint4[27968] = {X 105.1923, Y 47.9263, Z -6.3333, A 0.000, B 0.000, C 0.000 }
gfCNCPoint4[27969] = {X 104.6069, Y 48.4370, Z -6.3333, A 0.000, B 0.000, C 0.000 }
gfCNCPoint4[27970] = {X 103.9382, Y 48.8323, Z -6.3333, A 0.000, B 0.000, C 0.000 }
gfCNCPoint4[27971] = {X 103.0119, Y 49.1460, Z -6.3333, A 0.000, B 0.000, C 0.000 }
gfCNCPoint4[27972] = {X 102.0384, Y 49.2391, Z -6.3333, A 0.000, B 0.000, C 0.000 }
gfCNCPoint4[27973] = {X 101.0695, Y 49.1068, Z -6.3333, A 0.000, B 0.000, C 0.000 }
gfCNCPoint4[27974] = {X 100.1566, Y 48.7559, Z -6.3333, A 0.000, B 0.000, C 0.000 }
gfCNCPoint4[27975] = {X 99.3484, Y 48.2052, Z -6.3333, A 0.000, B 0.000, C 0.000 }
gfCNCPoint4[27976] = {X 98.6879, Y 47.4840, Z -6.3333, A 0.000, B 0.000, C 0.000 }
gfCNCPoint4[27977] = {X 98.2102, Y 46.6307, Z -6.3333, A 0.000, B 0.000, C 0.000 }
gfCNCPoint4[27978] = {X 95.0517, Y 38.9062, Z -6.3333, A 0.000, B 0.000, C 0.000 }
gfCNCPoint4[27979] = {X 95.0517, Y 40.9416, Z -6.3333, A 0.000, B 0.000, C 0.000 }
gfCNCPoint4[27980] = {X 95.5841, Y 41.4799, Z -6.3333, A 0.000, B 0.000, C 0.000 }
gfCNCPoint4[27981] = {X 96.0144, Y 42.1027, Z -6.3333, A 0.000, B 0.000, C 0.000 }
gfCNCPoint4[27982] = {X 96.2572, Y 42.6023, Z -6.3333, A 0.000, B 0.000, C 0.000 }
gfCNCPoint4[27983] = {X 96.4340, Y 43.1289, Z -6.3333, A 0.000, B 0.000, C 0.000 }
gfCNCPoint4[27984] = {X 96.5403, Y 43.6635, Z -6.3333, A 0.000, B 0.000, C 0.000 }
gfCNCPoint4[27985] = {X 96.5785, Y 44.2072, Z -6.3333, A 0.000, B 0.000, C 0.000 }
gfCNCPoint4[27986] = {X 96.5783, Y 45.0408, Z -6.3333, A 0.000, B 0.000, C 0.000 }
gfCNCPoint4[27987] = {X 96.4643, Y 45.9775, Z -6.3333, A 0.000, B 0.000, C 0.000 }
gfCNCPoint4[27988] = {X 96.1459, Y 46.8659, Z -6.3333, A 0.000, B 0.000, C 0.000 }
gfCNCPoint4[27989] = {X 95.6389, Y 47.6618, Z -6.3333, A 0.000, B 0.000, C 0.000 }
gfCNCPoint4[27990] = {X 94.9685, Y 48.3258, Z -6.3333, A 0.000, B 0.000, C 0.000 }
gfCNCPoint4[27991] = {X 94.1677, Y 48.8251, Z -6.3333, A 0.000, B 0.000, C 0.000 }
gfCNCPoint4[27992] = {X 93.2764, Y 49.1350, Z -6.3333, A 0.000, B 0.000, C 0.000 }
gfCNCPoint4[27993] = {X 92.3385, Y 49.2400, Z -6.3333, A 0.000, B 0.000, C 0.000 }
gfCNCPoint4[27994] = {X 85.8951, Y 49.2400, Z -6.3333, A 0.000, B 0.000, C 0.000 }
gfCNCPoint4[27995] = {X 84.9564, Y 49.1348, Z -6.3333, A 0.000, B 0.000, C 0.000 }
gfCNCPoint4[27996] = {X 84.0643, Y 48.8244, Z -6.3333, A 0.000, B 0.000, C 0.000 }
gfCNCPoint4[27997] = {X 83.2631, Y 48.3242, Z -6.3333, A 0.000, B 0.000, C 0.000 }
gfCNCPoint4[27998] = {X 82.5924, Y 47.6590, Z -6.3333, A 0.000, B 0.000, C 0.000 }
gfCNCPoint4[27999] = {X 82.0857, Y 46.8618, Z -6.3333, A 0.000, B 0.000, C 0.000 }
gfCNCPoint4[28000] = {X 81.7681, Y 45.9723, Z -6.3333, A 0.000, B 0.000, C 0.000 }
gfCNCPoint4[28001] = {X 81.6552, Y 45.0345, Z -6.3333, A 0.000, B 0.000, C 0.000 }
gfCNCPoint4[28002] = {X 81.6551, Y 44.2076, Z -6.3333, A 0.000, B 0.000, C 0.000 }
gfCNCPoint4[28003] = {X 81.7600, Y 43.2862, Z -6.3333, A 0.000, B 0.000, C 0.000 }
gfCNCPoint4[28004] = {X 82.0603, Y 42.4089, Z -6.3333, A 0.000, B 0.000, C 0.000 }
gfCNCPoint4[28005] = {X 82.5418, Y 41.6164, Z -6.3333, A 0.000, B 0.000, C 0.000 }
gfCNCPoint4[28006] = {X 83.1822, Y 40.9457, Z -6.3333, A 0.000, B 0.000, C 0.000 }
gfCNCPoint4[28007] = {X 83.1820, Y 28.5912, Z -6.3333, A 0.000, B 0.000, C 0.000 }
gfCNCPoint4[28008] = {X 79.1820, Y 28.5912, Z -6.3333, A 0.000, B 0.000, C 0.000 }
gfCNCPoint4[28009] = {X 83.2620, Y 28.5912, Z -6.3333, A 0.000, B 0.000, C 0.000 }
gfCNCPoint4[28010] = {X 83.2619, Y 16.1986, Z -6.3333, A 0.000, B 0.000, C 0.000 }
gfCNCPoint4[28011] = {X 82.6246, Y 15.5489, Z -6.3333, A 0.000, B 0.000, C 0.000 }
gfCNCPoint4[28012] = {X 82.1438, Y 14.7762, Z -6.3333, A 0.000, B 0.000, C 0.000 }
gfCNCPoint4[28013] = {X 81.8425, Y 13.9174, Z -6.3333, A 0.000, B 0.000, C 0.000 }
gfCNCPoint4[28014] = {X 81.7352, Y 13.0136, Z -6.3333, A 0.000, B 0.000, C 0.000 }
gfCNCPoint4[28015] = {X 81.7351, Y 12.1868, Z -6.3333, A 0.000, B 0.000, C 0.000 }
gfCNCPoint4[28016] = {X 81.8394, Y 11.2611, Z -6.3333, A 0.000, B 0.000, C 0.000 }
gfCNCPoint4[28017] = {X 82.1470, Y 10.3819, Z -6.3333, A 0.000, B 0.000, C 0.000 }
gfCNCPoint4[28018] = {X 82.6427, Y 9.5931, Z -6.3333, A 0.000, B 0.000, C 0.000 }
gfCNCPoint4[28019] = {X 83.3014, Y 8.9344, Z -6.3333, A 0.000, B 0.000, C 0.000 }
gfCNCPoint4[28020] = {X 84.0901, Y 8.4388, Z -6.3333, A 0.000, B 0.000, C 0.000 }
gfCNCPoint4[28021] = {X 84.9694, Y 8.1311, Z -6.3333, A 0.000, B 0.000, C 0.000 }
gfCNCPoint4[28022] = {X 85.8951, Y 8.0268, Z -6.3333, A 0.000, B 0.000, C 0.000 }
gfCNCPoint4[28023] = {X 94.0497, Y 8.0268, Z -6.3333, A 0.000, B 0.000, C 0.000 }
gfCNCPoint4[28024] = {X 94.9754, Y 8.1311, Z -6.3333, A 0.000, B 0.000, C 0.000 }
gfCNCPoint4[28025] = {X 95.8546, Y 8.4388, Z -6.3333, A 0.000, B 0.000, C 0.000 }
gfCNCPoint4[28026] = {X 96.6434, Y 8.9344, Z -6.3333, A 0.000, B 0.000, C 0.000 }
gfCNCPoint4[28027] = {X 97.3021, Y 9.5931, Z -6.3333, A 0.000, B 0.000, C 0.000 }
gfCNCPoint4[28028] = {X 97.7977, Y 10.3819, Z -6.3333, A 0.000, B 0.000, C 0.000 }
gfCNCPoint4[28029] = {X 98.1054, Y 11.2611, Z -6.3333, A 0.000, B 0.000, C 0.000 }
gfCNCPoint4[28030] = {X 98.2097, Y 12.1868, Z -6.3333, A 0.000, B 0.000, C 0.000 }
gfCNCPoint4[28031] = {X 98.2097, Y 12.9782, Z -6.3333, A 0.000, B 0.000, C 0.000 }
gfCNCPoint4[28032] = {X 98.1344, Y 13.7658, Z -6.3333, A 0.000, B 0.000, C 0.000 }
gfCNCPoint4[28033] = {X 97.9114, Y 14.5248, Z -6.3333, A 0.000, B 0.000, C 0.000 }
gfCNCPoint4[28034] = {X 97.5487, Y 15.2280, Z -6.3333, A 0.000, B 0.000, C 0.000 }
gfCNCPoint4[28035] = {X 101.8761, Y 25.9512, Z -6.3333, A 0.000, B 0.000, C 0.000 }
gfCNCPoint4[28036] = {X 106.1949, Y 15.2055, Z -6.3333, A 0.000, B 0.000, C 0.000 }
gfCNCPoint4[28037] = {X 105.8447, Y 14.5202, Z -6.3333, A 0.000, B 0.000, C 0.000 }
gfCNCPoint4[28038] = {X 105.6267, Y 13.7821, Z -6.3333, A 0.000, B 0.000, C 0.000 }
gfCNCPoint4[28039] = {X 105.5485, Y 13.0164, Z -6.3333, A 0.000, B 0.000, C 0.000 }
gfCNCPoint4[28040] = {X 105.5483, Y 12.1868, Z -6.3333, A 0.000, B 0.000, C 0.000 }
gfCNCPoint4[28041] = {X 105.6526, Y 11.2611, Z -6.3333, A 0.000, B 0.000, C 0.000 }
gfCNCPoint4[28042] = {X 105.9602, Y 10.3819, Z -6.3333, A 0.000, B 0.000, C 0.000 }
gfCNCPoint4[28043] = {X 106.4559, Y 9.5931, Z -6.3333, A 0.000, B 0.000, C 0.000 }
gfCNCPoint4[28044] = {X 107.1146, Y 8.9344, Z -6.3333, A 0.000, B 0.000, C 0.000 }
gfCNCPoint4[28045] = {X 107.9033, Y 8.4388, Z -6.3333, A 0.000, B 0.000, C 0.000 }
gfCNCPoint4[28046] = {X 108.7826, Y 8.1311, Z -6.3333, A 0.000, B 0.000, C 0.000 }
gfCNCPoint4[28047] = {X 109.7083, Y 8.0268, Z -6.3333, A 0.000, B 0.000, C 0.000 }
gfCNCPoint4[28048] = {X 117.7916, Y 8.0268, Z -6.3333, A 0.000, B 0.000, C 0.000 }
gfCNCPoint4[28049] = {X 118.7173, Y 8.1311, Z -6.3333, A 0.000, B 0.000, C 0.000 }
gfCNCPoint4[28050] = {X 119.5965, Y 8.4388, Z -6.3333, A 0.000, B 0.000, C 0.000 }
gfCNCPoint4[28051] = {X 120.3853, Y 8.9344, Z -6.3333, A 0.000, B 0.000, C 0.000 }
gfCNCPoint4[28052] = {X 121.0440, Y 9.5931, Z -6.3333, A 0.000, B 0.000, C 0.000 }
gfCNCPoint4[28053] = {X 121.5396, Y 10.3819, Z -6.3333, A 0.000, B 0.000, C 0.000 }
gfCNCPoint4[28054] = {X 121.8473, Y 11.2611, Z -6.3333, A 0.000, B 0.000, C 0.000 }
gfCNCPoint4[28055] = {X 121.9516, Y 12.1868, Z -6.3333, A 0.000, B 0.000, C 0.000 }
gfCNCPoint4[28056] = {X 121.9516, Y 12.9782, Z -6.3333, A 0.000, B 0.000, C 0.000 }
gfCNCPoint4[28057] = {X 121.8501, Y 13.8913, Z -6.3333, A 0.000, B 0.000, C 0.000 }
gfCNCPoint4[28058] = {X 121.5506, Y 14.7599, Z -6.3333, A 0.000, B 0.000, C 0.000 }
gfCNCPoint4[28059] = {X 121.0678, Y 15.5416, Z -6.3333, A 0.000, B 0.000, C 0.000 }
gfCNCPoint4[28060] = {X 120.4251, Y 16.1983, Z -6.3333, A 0.000, B 0.000, C 0.000 }
gfCNCPoint4[28061] = {X 120.4247, Y 40.9901, Z -6.3333, A 0.000, B 0.000, C 0.000 }
gfCNCPoint4[28062] = {X 120.5193, Y 41.0679, Z -6.3333, A 0.000, B 0.000, C 0.000 }
gfCNCPoint4[28063] = {X 121.1188, Y 41.7118, Z -6.3333, A 0.000, B 0.000, C 0.000 }
gfCNCPoint4[28064] = {X 121.5695, Y 42.4673, Z -6.3333, A 0.000, B 0.000, C 0.000 }
gfCNCPoint4[28065] = {X 121.8512, Y 43.3007, Z -6.3333, A 0.000, B 0.000, C 0.000 }
gfCNCPoint4[28066] = {X 121.9514, Y 44.1747, Z -6.3333, A 0.000, B 0.000, C 0.000 }
gfCNCPoint4[28067] = {X 121.9516, Y 45.0000, Z -6.3333, A 0.000, B 0.000, C 0.000 }
gfCNCPoint4[28068] = {X 121.8473, Y 45.9257, Z -6.3333, A 0.000, B 0.000, C 0.000 }
gfCNCPoint4[28069] = {X 121.5396, Y 46.8050, Z -6.3333, A 0.000, B 0.000, C 0.000 }
gfCNCPoint4[28070] = {X 121.0440, Y 47.5937, Z -6.3333, A 0.000, B 0.000, C 0.000 }
gfCNCPoint4[28071] = {X 120.3853, Y 48.2524, Z -6.3333, A 0.000, B 0.000, C 0.000 }
gfCNCPoint4[28072] = {X 119.5965, Y 48.7480, Z -6.3333, A 0.000, B 0.000, C 0.000 }
gfCNCPoint4[28073] = {X 118.7173, Y 49.0557, Z -6.3333, A 0.000, B 0.000, C 0.000 }
gfCNCPoint4[28074] = {X 117.7916, Y 49.1600, Z -6.3333, A 0.000, B 0.000, C 0.000 }
gfCNCPoint4[28075] = {X 111.9185, Y 49.1600, Z -6.3333, A 0.000, B 0.000, C 0.000 }
gfCNCPoint4[28076] = {X 110.9974, Y 49.0567, Z -6.3333, A 0.000, B 0.000, C 0.000 }
gfCNCPoint4[28077] = {X 110.1220, Y 48.7521, Z -6.3333, A 0.000, B 0.000, C 0.000 }
gfCNCPoint4[28078] = {X 109.3358, Y 48.2612, Z -6.3333, A 0.000, B 0.000, C 0.000 }
gfCNCPoint4[28079] = {X 108.6778, Y 47.6084, Z -6.3333, A 0.000, B 0.000, C 0.000 }
gfCNCPoint4[28080] = {X 108.1807, Y 46.8261, Z -6.3333, A 0.000, B 0.000, C 0.000 }
gfCNCPoint4[28081] = {X 107.8691, Y 45.9531, Z -6.3333, A 0.000, B 0.000, C 0.000 }
gfCNCPoint4[28082] = {X 107.7586, Y 45.0328, Z -6.3333, A 0.000, B 0.000, C 0.000 }
gfCNCPoint4[28083] = {X 107.7585, Y 44.1789, Z -6.3333, A 0.000, B 0.000, C 0.000 }
gfCNCPoint4[28084] = {X 107.7927, Y 43.6574, Z -6.3333, A 0.000, B 0.000, C 0.000 }
gfCNCPoint4[28085] = {X 107.8946, Y 43.1449, Z -6.3333, A 0.000, B 0.000, C 0.000 }
gfCNCPoint4[28086] = {X 108.0562, Y 42.6653, Z -6.3333, A 0.000, B 0.000, C 0.000 }
gfCNCPoint4[28087] = {X 108.2772, Y 42.2099, Z -6.3333, A 0.000, B 0.000, C 0.000 }
gfCNCPoint4[28088] = {X 108.7349, Y 41.5337, Z -6.3333, A 0.000, B 0.000, C 0.000 }
gfCNCPoint4[28089] = {X 109.2853, Y 40.9305, Z -6.3333, A 0.000, B 0.000, C 0.000 }
gfCNCPoint4[28090] = {X 109.2851, Y 39.0829, Z -6.3333, A 0.000, B 0.000, C 0.000 }
gfCNCPoint4[28091] = {X 109.0402, Y 39.0829, Z -6.3333, A 0.000, B 0.000, C 0.000 }
gfCNCPoint4[28092] = {X 105.9641, Y 46.5999, Z -6.3333, A 0.000, B 0.000, C 0.000 }
gfCNCPoint4[28093] = {X 105.6077, Y 47.2737, Z -6.3333, A 0.000, B 0.000, C 0.000 }
gfCNCPoint4[28094] = {X 105.1344, Y 47.8711, Z -6.3333, A 0.000, B 0.000, C 0.000 }
gfCNCPoint4[28095] = {X 104.5601, Y 48.3721, Z -6.3333, A 0.000, B 0.000, C 0.000 }
gfCNCPoint4[28096] = {X 103.9040, Y 48.7600, Z -6.3333, A 0.000, B 0.000, C 0.000 }
gfCNCPoint4[28097] = {X 102.9952, Y 49.0678, Z -6.3333, A 0.000, B 0.000, C 0.000 }
gfCNCPoint4[28098] = {X 102.0400, Y 49.1592, Z -6.3333, A 0.000, B 0.000, C 0.000 }
gfCNCPoint4[28099] = {X 101.0894, Y 49.0293, Z -6.3333, A 0.000, B 0.000, C 0.000 }
gfCNCPoint4[28100] = {X 100.1937, Y 48.6850, Z -6.3333, A 0.000, B 0.000, C 0.000 }
gfCNCPoint4[28101] = {X 99.4008, Y 48.1448, Z -6.3333, A 0.000, B 0.000, C 0.000 }
gfCNCPoint4[28102] = {X 98.7527, Y 47.4372, Z -6.3333, A 0.000, B 0.000, C 0.000 }
gfCNCPoint4[28103] = {X 98.2840, Y 46.5999, Z -6.3333, A 0.000, B 0.000, C 0.000 }
gfCNCPoint4[28104] = {X 94.9716, Y 38.4992, Z -6.3333, A 0.000, B 0.000, C 0.000 }
gfCNCPoint4[28105] = {X 94.9717, Y 40.9789, Z -6.3333, A 0.000, B 0.000, C 0.000 }
gfCNCPoint4[28106] = {X 95.5107, Y 41.5167, Z -6.3333, A 0.000, B 0.000, C 0.000 }
gfCNCPoint4[28107] = {X 95.9448, Y 42.1423, Z -6.3333, A 0.000, B 0.000, C 0.000 }
gfCNCPoint4[28108] = {X 96.1832, Y 42.6326, Z -6.3333, A 0.000, B 0.000, C 0.000 }
gfCNCPoint4[28109] = {X 96.3567, Y 43.1495, Z -6.3333, A 0.000, B 0.000, C 0.000 }
gfCNCPoint4[28110] = {X 96.4610, Y 43.6741, Z -6.3333, A 0.000, B 0.000, C 0.000 }
gfCNCPoint4[28111] = {X 96.4985, Y 44.2077, Z -6.3333, A 0.000, B 0.000, C 0.000 }
gfCNCPoint4[28112] = {X 96.4983, Y 45.0400, Z -6.3333, A 0.000, B 0.000, C 0.000 }
gfCNCPoint4[28113] = {X 96.3865, Y 45.9591, Z -6.3333, A 0.000, B 0.000, C 0.000 }
gfCNCPoint4[28114] = {X 96.0741, Y 46.8306, Z -6.3333, A 0.000, B 0.000, C 0.000 }
gfCNCPoint4[28115] = {X 95.5767, Y 47.6115, Z -6.3333, A 0.000, B 0.000, C 0.000 }
gfCNCPoint4[28116] = {X 94.9188, Y 48.2631, Z -6.3333, A 0.000, B 0.000, C 0.000 }
gfCNCPoint4[28117] = {X 94.1332, Y 48.7530, Z -6.3333, A 0.000, B 0.000, C 0.000 }
gfCNCPoint4[28118] = {X 93.2587, Y 49.0570, Z -6.3333, A 0.000, B 0.000, C 0.000 }
gfCNCPoint4[28119] = {X 92.3385, Y 49.1600, Z -6.3333, A 0.000, B 0.000, C 0.000 }
gfCNCPoint4[28120] = {X 85.8951, Y 49.1600, Z -6.3333, A 0.000, B 0.000, C 0.000 }
gfCNCPoint4[28121] = {X 84.9741, Y 49.0568, Z -6.3333, A 0.000, B 0.000, C 0.000 }
gfCNCPoint4[28122] = {X 84.0988, Y 48.7522, Z -6.3333, A 0.000, B 0.000, C 0.000 }
gfCNCPoint4[28123] = {X 83.3127, Y 48.2614, Z -6.3333, A 0.000, B 0.000, C 0.000 }
gfCNCPoint4[28124] = {X 82.6547, Y 47.6088, Z -6.3333, A 0.000, B 0.000, C 0.000 }
gfCNCPoint4[28125] = {X 82.1576, Y 46.8267, Z -6.3333, A 0.000, B 0.000, C 0.000 }
gfCNCPoint4[28126] = {X 81.8459, Y 45.9539, Z -6.3333, A 0.000, B 0.000, C 0.000 }
gfCNCPoint4[28127] = {X 81.7352, Y 45.0338, Z -6.3333, A 0.000, B 0.000, C 0.000 }
gfCNCPoint4[28128] = {X 81.7351, Y 44.2080, Z -6.3333, A 0.000, B 0.000, C 0.000 }
gfCNCPoint4[28129] = {X 81.8401, Y 43.2948, Z -6.3333, A 0.000, B 0.000, C 0.000 }
gfCNCPoint4[28130] = {X 82.1406, Y 42.4260, Z -6.3333, A 0.000, B 0.000, C 0.000 }
gfCNCPoint4[28131] = {X 82.6223, Y 41.6431, Z -6.3333, A 0.000, B 0.000, C 0.000 }
gfCNCPoint4[28132] = {X 83.2622, Y 40.9832, Z -6.3333, A 0.000, B 0.000, C 0.000 }
gfCNCPoint4[28133] = {X 83.2620, Y 28.5912, Z -6.3333, A 0.000, B 0.000, C 0.000 }
gfCNCPoint4[28134] = {X 79.2620, Y 28.5912, Z -6.3333, A 0.000, B 0.000, C 0.000 }
gfCNCPoint4[28135] = {X 83.3420, Y 28.5912, Z -6.3333, A 0.000, B 0.000, C 0.000 }
gfCNCPoint4[28136] = {X 83.3419, Y 16.1604, Z -6.3333, A 0.000, B 0.000, C 0.000 }
gfCNCPoint4[28137] = {X 82.7051, Y 15.5217, Z -6.3333, A 0.000, B 0.000, C 0.000 }
gfCNCPoint4[28138] = {X 82.2241, Y 14.7586, Z -6.3333, A 0.000, B 0.000, C 0.000 }
gfCNCPoint4[28139] = {X 81.9226, Y 13.9085, Z -6.3333, A 0.000, B 0.000, C 0.000 }
gfCNCPoint4[28140] = {X 81.8152, Y 13.0129, Z -6.3333, A 0.000, B 0.000, C 0.000 }
gfCNCPoint4[28141] = {X 81.8151, Y 12.1868, Z -6.3333, A 0.000, B 0.000, C 0.000 }
gfCNCPoint4[28142] = {X 81.9174, Y 11.2789, Z -6.3333, A 0.000, B 0.000, C 0.000 }
gfCNCPoint4[28143] = {X 82.2191, Y 10.4166, Z -6.3333, A 0.000, B 0.000, C 0.000 }
gfCNCPoint4[28144] = {X 82.7052, Y 9.6430, Z -6.3333, A 0.000, B 0.000, C 0.000 }
gfCNCPoint4[28145] = {X 83.3512, Y 8.9969, Z -6.3333, A 0.000, B 0.000, C 0.000 }
gfCNCPoint4[28146] = {X 84.1248, Y 8.5109, Z -6.3333, A 0.000, B 0.000, C 0.000 }
gfCNCPoint4[28147] = {X 84.9872, Y 8.2091, Z -6.3333, A 0.000, B 0.000, C 0.000 }
gfCNCPoint4[28148] = {X 85.8951, Y 8.1068, Z -6.3333, A 0.000, B 0.000, C 0.000 }
gfCNCPoint4[28149] = {X 94.0497, Y 8.1068, Z -6.3333, A 0.000, B 0.000, C 0.000 }
gfCNCPoint4[28150] = {X 94.9576, Y 8.2091, Z -6.3333, A 0.000, B 0.000, C 0.000 }
gfCNCPoint4[28151] = {X 95.8199, Y 8.5109, Z -6.3333, A 0.000, B 0.000, C 0.000 }
gfCNCPoint4[28152] = {X 96.5935, Y 8.9969, Z -6.3333, A 0.000, B 0.000, C 0.000 }
gfCNCPoint4[28153] = {X 97.2395, Y 9.6430, Z -6.3333, A 0.000, B 0.000, C 0.000 }
gfCNCPoint4[28154] = {X 97.7256, Y 10.4166, Z -6.3333, A 0.000, B 0.000, C 0.000 }
gfCNCPoint4[28155] = {X 98.0274, Y 11.2789, Z -6.3333, A 0.000, B 0.000, C 0.000 }
gfCNCPoint4[28156] = {X 98.1297, Y 12.1868, Z -6.3333, A 0.000, B 0.000, C 0.000 }
gfCNCPoint4[28157] = {X 98.1297, Y 12.9782, Z -6.3333, A 0.000, B 0.000, C 0.000 }
gfCNCPoint4[28158] = {X 98.0632, Y 13.7118, Z -6.3333, A 0.000, B 0.000, C 0.000 }
gfCNCPoint4[28159] = {X 97.8658, Y 14.4214, Z -6.3333, A 0.000, B 0.000, C 0.000 }
gfCNCPoint4[28160] = {X 97.5441, Y 15.0841, Z -6.3333, A 0.000, B 0.000, C 0.000 }
gfCNCPoint4[28161] = {X 97.4976, Y 15.1594, Z -6.3333, A 0.000, B 0.000, C 0.000 }
gfCNCPoint4[28162] = {X 97.4494, Y 15.2337, Z -6.3333, A 0.000, B 0.000, C 0.000 }
gfCNCPoint4[28163] = {X 97.4861, Y 15.2810, Z -6.3333, A 0.000, B 0.000, C 0.000 }
gfCNCPoint4[28164] = {X 101.8762, Y 26.1654, Z -6.3333, A 0.000, B 0.000, C 0.000 }
gfCNCPoint4[28165] = {X 106.2845, Y 15.1970, Z -6.3333, A 0.000, B 0.000, C 0.000 }
gfCNCPoint4[28166] = {X 106.2410, Y 15.1284, Z -6.3333, A 0.000, B 0.000, C 0.000 }
gfCNCPoint4[28167] = {X 106.1988, Y 15.0589, Z -6.3333, A 0.000, B 0.000, C 0.000 }
gfCNCPoint4[28168] = {X 105.8897, Y 14.4149, Z -6.3333, A 0.000, B 0.000, C 0.000 }
gfCNCPoint4[28169] = {X 105.6976, Y 13.7268, Z -6.3333, A 0.000, B 0.000, C 0.000 }
gfCNCPoint4[28170] = {X 105.6285, Y 13.0157, Z -6.3333, A 0.000, B 0.000, C 0.000 }
gfCNCPoint4[28171] = {X 105.6283, Y 12.1868, Z -6.3333, A 0.000, B 0.000, C 0.000 }
gfCNCPoint4[28172] = {X 105.7306, Y 11.2789, Z -6.3333, A 0.000, B 0.000, C 0.000 }
gfCNCPoint4[28173] = {X 106.0323, Y 10.4166, Z -6.3333, A 0.000, B 0.000, C 0.000 }
gfCNCPoint4[28174] = {X 106.5184, Y 9.6430, Z -6.3333, A 0.000, B 0.000, C 0.000 }
gfCNCPoint4[28175] = {X 107.1644, Y 8.9969, Z -6.3333, A 0.000, B 0.000, C 0.000 }
gfCNCPoint4[28176] = {X 107.9380, Y 8.5109, Z -6.3333, A 0.000, B 0.000, C 0.000 }
gfCNCPoint4[28177] = {X 108.8004, Y 8.2091, Z -6.3333, A 0.000, B 0.000, C 0.000 }
gfCNCPoint4[28178] = {X 109.7083, Y 8.1068, Z -6.3333, A 0.000, B 0.000, C 0.000 }
gfCNCPoint4[28179] = {X 117.7916, Y 8.1068, Z -6.3333, A 0.000, B 0.000, C 0.000 }
gfCNCPoint4[28180] = {X 118.6995, Y 8.2091, Z -6.3333, A 0.000, B 0.000, C 0.000 }
gfCNCPoint4[28181] = {X 119.5618, Y 8.5109, Z -6.3333, A 0.000, B 0.000, C 0.000 }
gfCNCPoint4[28182] = {X 120.3354, Y 8.9969, Z -6.3333, A 0.000, B 0.000, C 0.000 }
gfCNCPoint4[28183] = {X 120.9814, Y 9.6430, Z -6.3333, A 0.000, B 0.000, C 0.000 }
gfCNCPoint4[28184] = {X 121.4675, Y 10.4166, Z -6.3333, A 0.000, B 0.000, C 0.000 }
gfCNCPoint4[28185] = {X 121.7693, Y 11.2789, Z -6.3333, A 0.000, B 0.000, C 0.000 }
gfCNCPoint4[28186] = {X 121.8716, Y 12.1868, Z -6.3333, A 0.000, B 0.000, C 0.000 }
gfCNCPoint4[28187] = {X 121.8716, Y 12.9782, Z -6.3333, A 0.000, B 0.000, C 0.000 }
gfCNCPoint4[28188] = {X 121.7699, Y 13.8830, Z -6.3333, A 0.000, B 0.000, C 0.000 }
gfCNCPoint4[28189] = {X 121.4702, Y 14.7427, Z -6.3333, A 0.000, B 0.000, C 0.000 }
gfCNCPoint4[28190] = {X 120.9872, Y 15.5146, Z -6.3333, A 0.000, B 0.000, C 0.000 }
gfCNCPoint4[28191] = {X 120.3451, Y 16.1601, Z -6.3333, A 0.000, B 0.000, C 0.000 }
gfCNCPoint4[28192] = {X 120.3447, Y 41.0278, Z -6.3333, A 0.000, B 0.000, C 0.000 }
gfCNCPoint4[28193] = {X 120.4677, Y 41.1290, Z -6.3333, A 0.000, B 0.000, C 0.000 }
gfCNCPoint4[28194] = {X 121.0553, Y 41.7604, Z -6.3333, A 0.000, B 0.000, C 0.000 }
gfCNCPoint4[28195] = {X 121.4971, Y 42.5013, Z -6.3333, A 0.000, B 0.000, C 0.000 }
gfCNCPoint4[28196] = {X 121.7732, Y 43.3184, Z -6.3333, A 0.000, B 0.000, C 0.000 }
gfCNCPoint4[28197] = {X 121.8714, Y 44.1754, Z -6.3333, A 0.000, B 0.000, C 0.000 }
gfCNCPoint4[28198] = {X 121.8716, Y 45.0000, Z -6.3333, A 0.000, B 0.000, C 0.000 }
gfCNCPoint4[28199] = {X 121.7693, Y 45.9079, Z -6.3333, A 0.000, B 0.000, C 0.000 }
gfCNCPoint4[28200] = {X 121.4675, Y 46.7702, Z -6.3333, A 0.000, B 0.000, C 0.000 }
gfCNCPoint4[28201] = {X 120.9814, Y 47.5438, Z -6.3333, A 0.000, B 0.000, C 0.000 }
gfCNCPoint4[28202] = {X 120.3354, Y 48.1899, Z -6.3333, A 0.000, B 0.000, C 0.000 }
gfCNCPoint4[28203] = {X 119.5618, Y 48.6760, Z -6.3333, A 0.000, B 0.000, C 0.000 }
gfCNCPoint4[28204] = {X 118.6995, Y 48.9777, Z -6.3333, A 0.000, B 0.000, C 0.000 }
gfCNCPoint4[28205] = {X 117.7916, Y 49.0800, Z -6.3333, A 0.000, B 0.000, C 0.000 }
gfCNCPoint4[28206] = {X 111.9185, Y 49.0800, Z -6.3333, A 0.000, B 0.000, C 0.000 }
gfCNCPoint4[28207] = {X 111.0151, Y 48.9787, Z -6.3333, A 0.000, B 0.000, C 0.000 }
gfCNCPoint4[28208] = {X 110.1565, Y 48.6799, Z -6.3333, A 0.000, B 0.000, C 0.000 }
gfCNCPoint4[28209] = {X 109.3855, Y 48.1985, Z -6.3333, A 0.000, B 0.000, C 0.000 }
gfCNCPoint4[28210] = {X 108.7401, Y 47.5582, Z -6.3333, A 0.000, B 0.000, C 0.000 }
gfCNCPoint4[28211] = {X 108.2526, Y 46.7909, Z -6.3333, A 0.000, B 0.000, C 0.000 }
gfCNCPoint4[28212] = {X 107.9470, Y 45.9348, Z -6.3333, A 0.000, B 0.000, C 0.000 }
gfCNCPoint4[28213] = {X 107.8386, Y 45.0322, Z -6.3333, A 0.000, B 0.000, C 0.000 }
gfCNCPoint4[28214] = {X 107.8385, Y 44.1789, Z -6.3333, A 0.000, B 0.000, C 0.000 }
gfCNCPoint4[28215] = {X 107.8720, Y 43.6679, Z -6.3333, A 0.000, B 0.000, C 0.000 }
gfCNCPoint4[28216] = {X 107.9718, Y 43.1656, Z -6.3333, A 0.000, B 0.000, C 0.000 }
gfCNCPoint4[28217] = {X 108.1302, Y 42.6956, Z -6.3333, A 0.000, B 0.000, C 0.000 }
gfCNCPoint4[28218] = {X 108.3468, Y 42.2493, Z -6.3333, A 0.000, B 0.000, C 0.000 }
gfCNCPoint4[28219] = {X 108.8086, Y 41.5696, Z -6.3333, A 0.000, B 0.000, C 0.000 }
gfCNCPoint4[28220] = {X 109.3653, Y 40.9650, Z -6.3333, A 0.000, B 0.000, C 0.000 }
gfCNCPoint4[28221] = {X 109.3651, Y 39.0029, Z -6.3333, A 0.000, B 0.000, C 0.000 }
gfCNCPoint4[28222] = {X 108.9865, Y 39.0029, Z -6.3333, A 0.000, B 0.000, C 0.000 }
gfCNCPoint4[28223] = {X 105.8902, Y 46.5692, Z -6.3333, A 0.000, B 0.000, C 0.000 }
gfCNCPoint4[28224] = {X 105.5407, Y 47.2300, Z -6.3333, A 0.000, B 0.000, C 0.000 }
gfCNCPoint4[28225] = {X 105.0765, Y 47.8159, Z -6.3333, A 0.000, B 0.000, C 0.000 }
gfCNCPoint4[28226] = {X 104.5133, Y 48.3073, Z -6.3333, A 0.000, B 0.000, C 0.000 }
gfCNCPoint4[28227] = {X 103.8698, Y 48.6877, Z -6.3333, A 0.000, B 0.000, C 0.000 }
gfCNCPoint4[28228] = {X 102.9784, Y 48.9895, Z -6.3333, A 0.000, B 0.000, C 0.000 }
gfCNCPoint4[28229] = {X 102.0417, Y 49.0792, Z -6.3333, A 0.000, B 0.000, C 0.000 }
gfCNCPoint4[28230] = {X 101.1093, Y 48.9518, Z -6.3333, A 0.000, B 0.000, C 0.000 }
gfCNCPoint4[28231] = {X 100.2309, Y 48.6142, Z -6.3333, A 0.000, B 0.000, C 0.000 }
gfCNCPoint4[28232] = {X 99.4532, Y 48.0843, Z -6.3333, A 0.000, B 0.000, C 0.000 }
gfCNCPoint4[28233] = {X 98.8176, Y 47.3903, Z -6.3333, A 0.000, B 0.000, C 0.000 }
gfCNCPoint4[28234] = {X 98.3579, Y 46.5692, Z -6.3333, A 0.000, B 0.000, C 0.000 }
gfCNCPoint4[28235] = {X 94.8926, Y 38.0945, Z -6.3333, A 0.000, B 0.000, C 0.000 }
gfCNCPoint4[28236] = {X 94.8916, Y 38.2309, Z -6.3333, A 0.000, B 0.000, C 0.000 }
gfCNCPoint4[28237] = {X 94.8917, Y 41.0166, Z -6.3333, A 0.000, B 0.000, C 0.000 }
gfCNCPoint4[28238] = {X 95.4373, Y 41.5538, Z -6.3333, A 0.000, B 0.000, C 0.000 }
gfCNCPoint4[28239] = {X 95.8753, Y 42.1818, Z -6.3333, A 0.000, B 0.000, C 0.000 }
gfCNCPoint4[28240] = {X 96.1091, Y 42.6629, Z -6.3333, A 0.000, B 0.000, C 0.000 }
gfCNCPoint4[28241] = {X 96.2793, Y 43.1700, Z -6.3333, A 0.000, B 0.000, C 0.000 }
gfCNCPoint4[28242] = {X 96.3817, Y 43.6847, Z -6.3333, A 0.000, B 0.000, C 0.000 }
gfCNCPoint4[28243] = {X 96.4185, Y 44.2083, Z -6.3333, A 0.000, B 0.000, C 0.000 }
gfCNCPoint4[28244] = {X 96.4184, Y 45.0392, Z -6.3333, A 0.000, B 0.000, C 0.000 }
gfCNCPoint4[28245] = {X 96.3086, Y 45.9406, Z -6.3333, A 0.000, B 0.000, C 0.000 }
gfCNCPoint4[28246] = {X 96.0023, Y 46.7954, Z -6.3333, A 0.000, B 0.000, C 0.000 }
gfCNCPoint4[28247] = {X 95.5144, Y 47.5613, Z -6.3333, A 0.000, B 0.000, C 0.000 }
gfCNCPoint4[28248] = {X 94.8692, Y 48.2003, Z -6.3333, A 0.000, B 0.000, C 0.000 }
gfCNCPoint4[28249] = {X 94.0987, Y 48.6808, Z -6.3333, A 0.000, B 0.000, C 0.000 }
gfCNCPoint4[28250] = {X 93.2410, Y 48.9789, Z -6.3333, A 0.000, B 0.000, C 0.000 }
gfCNCPoint4[28251] = {X 92.3385, Y 49.0800, Z -6.3333, A 0.000, B 0.000, C 0.000 }
gfCNCPoint4[28252] = {X 85.8951, Y 49.0800, Z -6.3333, A 0.000, B 0.000, C 0.000 }
gfCNCPoint4[28253] = {X 84.9918, Y 48.9788, Z -6.3333, A 0.000, B 0.000, C 0.000 }
gfCNCPoint4[28254] = {X 84.1334, Y 48.6801, Z -6.3333, A 0.000, B 0.000, C 0.000 }
gfCNCPoint4[28255] = {X 83.3624, Y 48.1987, Z -6.3333, A 0.000, B 0.000, C 0.000 }
gfCNCPoint4[28256] = {X 82.7171, Y 47.5586, Z -6.3333, A 0.000, B 0.000, C 0.000 }
gfCNCPoint4[28257] = {X 82.2295, Y 46.7916, Z -6.3333, A 0.000, B 0.000, C 0.000 }
gfCNCPoint4[28258] = {X 81.9238, Y 45.9356, Z -6.3333, A 0.000, B 0.000, C 0.000 }
gfCNCPoint4[28259] = {X 81.8152, Y 45.0332, Z -6.3333, A 0.000, B 0.000, C 0.000 }
gfCNCPoint4[28260] = {X 81.8151, Y 44.2084, Z -6.3333, A 0.000, B 0.000, C 0.000 }
gfCNCPoint4[28261] = {X 81.9202, Y 43.3034, Z -6.3333, A 0.000, B 0.000, C 0.000 }
gfCNCPoint4[28262] = {X 82.2210, Y 42.4434, Z -6.3333, A 0.000, B 0.000, C 0.000 }
gfCNCPoint4[28263] = {X 82.7028, Y 41.6700, Z -6.3333, A 0.000, B 0.000, C 0.000 }
gfCNCPoint4[28264] = {X 83.3422, Y 41.0210, Z -6.3333, A 0.000, B 0.000, C 0.000 }
gfCNCPoint4[28265] = {X 83.3420, Y 28.5912, Z -6.3333, A 0.000, B 0.000, C 0.000 }
gfCNCPoint4[28266] = {X 79.3420, Y 28.5912, Z -6.3333, A 0.000, B 0.000, C 0.000 }
gfCNCPoint4[28267] = {X 83.4220, Y 28.5912, Z -6.3333, A 0.000, B 0.000, C 0.000 }
gfCNCPoint4[28268] = {X 83.4219, Y 16.1218, Z -6.3333, A 0.000, B 0.000, C 0.000 }
gfCNCPoint4[28269] = {X 82.7802, Y 15.4875, Z -6.3333, A 0.000, B 0.000, C 0.000 }
gfCNCPoint4[28270] = {X 82.2970, Y 14.7255, Z -6.3333, A 0.000, B 0.000, C 0.000 }
gfCNCPoint4[28271] = {X 81.9968, Y 13.8745, Z -6.3333, A 0.000, B 0.000, C 0.000 }
gfCNCPoint4[28272] = {X 81.8951, Y 12.9780, Z -6.3333, A 0.000, B 0.000, C 0.000 }
gfCNCPoint4[28273] = {X 81.8951, Y 12.1868, Z -6.3333, A 0.000, B 0.000, C 0.000 }
gfCNCPoint4[28274] = {X 81.9954, Y 11.2967, Z -6.3333, A 0.000, B 0.000, C 0.000 }
gfCNCPoint4[28275] = {X 82.2912, Y 10.4513, Z -6.3333, A 0.000, B 0.000, C 0.000 }
gfCNCPoint4[28276] = {X 82.7677, Y 9.6929, Z -6.3333, A 0.000, B 0.000, C 0.000 }
gfCNCPoint4[28277] = {X 83.4011, Y 9.0595, Z -6.3333, A 0.000, B 0.000, C 0.000 }
gfCNCPoint4[28278] = {X 84.1595, Y 8.5829, Z -6.3333, A 0.000, B 0.000, C 0.000 }
gfCNCPoint4[28279] = {X 85.0050, Y 8.2871, Z -6.3333, A 0.000, B 0.000, C 0.000 }
gfCNCPoint4[28280] = {X 85.8951, Y 8.1868, Z -6.3333, A 0.000, B 0.000, C 0.000 }
gfCNCPoint4[28281] = {X 94.0497, Y 8.1868, Z -6.3333, A 0.000, B 0.000, C 0.000 }
gfCNCPoint4[28282] = {X 94.9398, Y 8.2871, Z -6.3333, A 0.000, B 0.000, C 0.000 }
gfCNCPoint4[28283] = {X 95.7852, Y 8.5829, Z -6.3333, A 0.000, B 0.000, C 0.000 }
gfCNCPoint4[28284] = {X 96.5436, Y 9.0595, Z -6.3333, A 0.000, B 0.000, C 0.000 }
gfCNCPoint4[28285] = {X 97.1770, Y 9.6929, Z -6.3333, A 0.000, B 0.000, C 0.000 }
gfCNCPoint4[28286] = {X 97.6535, Y 10.4513, Z -6.3333, A 0.000, B 0.000, C 0.000 }
gfCNCPoint4[28287] = {X 97.9494, Y 11.2967, Z -6.3333, A 0.000, B 0.000, C 0.000 }
gfCNCPoint4[28288] = {X 98.0497, Y 12.1868, Z -6.3333, A 0.000, B 0.000, C 0.000 }
gfCNCPoint4[28289] = {X 98.0495, Y 13.0192, Z -6.3333, A 0.000, B 0.000, C 0.000 }
gfCNCPoint4[28290] = {X 97.9794, Y 13.7243, Z -6.3333, A 0.000, B 0.000, C 0.000 }
gfCNCPoint4[28291] = {X 97.7861, Y 14.4059, Z -6.3333, A 0.000, B 0.000, C 0.000 }
gfCNCPoint4[28292] = {X 97.4756, Y 15.0428, Z -6.3333, A 0.000, B 0.000, C 0.000 }
gfCNCPoint4[28293] = {X 97.4131, Y 15.1431, Z -6.3333, A 0.000, B 0.000, C 0.000 }
gfCNCPoint4[28294] = {X 97.3476, Y 15.2415, Z -6.3333, A 0.000, B 0.000, C 0.000 }
gfCNCPoint4[28295] = {X 97.4118, Y 15.3109, Z -6.3333, A 0.000, B 0.000, C 0.000 }
gfCNCPoint4[28296] = {X 97.9975, Y 16.7687, Z -6.3333, A 0.000, B 0.000, C 0.000 }
gfCNCPoint4[28297] = {X 101.6283, Y 25.7689, Z -6.3333, A 0.000, B 0.000, C 0.000 }
gfCNCPoint4[28298] = {X 101.8768, Y 26.3788, Z -6.3333, A 0.000, B 0.000, C 0.000 }
gfCNCPoint4[28299] = {X 104.7195, Y 19.2954, Z -6.3333, A 0.000, B 0.000, C 0.000 }
gfCNCPoint4[28300] = {X 106.3413, Y 15.2554, Z -6.3333, A 0.000, B 0.000, C 0.000 }
gfCNCPoint4[28301] = {X 106.3813, Y 15.1986, Z -6.3333, A 0.000, B 0.000, C 0.000 }
gfCNCPoint4[28302] = {X 106.3232, Y 15.1091, Z -6.3333, A 0.000, B 0.000, C 0.000 }
gfCNCPoint4[28303] = {X 106.2676, Y 15.0181, Z -6.3333, A 0.000, B 0.000, C 0.000 }
gfCNCPoint4[28304] = {X 105.9602, Y 14.3751, Z -6.3333, A 0.000, B 0.000, C 0.000 }
gfCNCPoint4[28305] = {X 105.7718, Y 13.6878, Z -6.3333, A 0.000, B 0.000, C 0.000 }
gfCNCPoint4[28306] = {X 105.7083, Y 12.9780, Z -6.3333, A 0.000, B 0.000, C 0.000 }
gfCNCPoint4[28307] = {X 105.7083, Y 12.1868, Z -6.3333, A 0.000, B 0.000, C 0.000 }
gfCNCPoint4[28308] = {X 105.8086, Y 11.2967, Z -6.3333, A 0.000, B 0.000, C 0.000 }
gfCNCPoint4[28309] = {X 106.1044, Y 10.4513, Z -6.3333, A 0.000, B 0.000, C 0.000 }
gfCNCPoint4[28310] = {X 106.5810, Y 9.6929, Z -6.3333, A 0.000, B 0.000, C 0.000 }
gfCNCPoint4[28311] = {X 107.2143, Y 9.0595, Z -6.3333, A 0.000, B 0.000, C 0.000 }
gfCNCPoint4[28312] = {X 107.9727, Y 8.5829, Z -6.3333, A 0.000, B 0.000, C 0.000 }
gfCNCPoint4[28313] = {X 108.8182, Y 8.2871, Z -6.3333, A 0.000, B 0.000, C 0.000 }
gfCNCPoint4[28314] = {X 109.7083, Y 8.1868, Z -6.3333, A 0.000, B 0.000, C 0.000 }
gfCNCPoint4[28315] = {X 117.7916, Y 8.1868, Z -6.3333, A 0.000, B 0.000, C 0.000 }
gfCNCPoint4[28316] = {X 118.6817, Y 8.2871, Z -6.3333, A 0.000, B 0.000, C 0.000 }
gfCNCPoint4[28317] = {X 119.5271, Y 8.5829, Z -6.3333, A 0.000, B 0.000, C 0.000 }
gfCNCPoint4[28318] = {X 120.2855, Y 9.0595, Z -6.3333, A 0.000, B 0.000, C 0.000 }
gfCNCPoint4[28319] = {X 120.9189, Y 9.6929, Z -6.3333, A 0.000, B 0.000, C 0.000 }
gfCNCPoint4[28320] = {X 121.3955, Y 10.4513, Z -6.3333, A 0.000, B 0.000, C 0.000 }
gfCNCPoint4[28321] = {X 121.6913, Y 11.2967, Z -6.3333, A 0.000, B 0.000, C 0.000 }
gfCNCPoint4[28322] = {X 121.7916, Y 12.1868, Z -6.3333, A 0.000, B 0.000, C 0.000 }
gfCNCPoint4[28323] = {X 121.7914, Y 13.0192, Z -6.3333, A 0.000, B 0.000, C 0.000 }
gfCNCPoint4[28324] = {X 121.6828, Y 13.9045, Z -6.3333, A 0.000, B 0.000, C 0.000 }
gfCNCPoint4[28325] = {X 121.3807, Y 14.7438, Z -6.3333, A 0.000, B 0.000, C 0.000 }
gfCNCPoint4[28326] = {X 120.9002, Y 15.4952, Z -6.3333, A 0.000, B 0.000, C 0.000 }
gfCNCPoint4[28327] = {X 120.2651, Y 16.1215, Z -6.3333, A 0.000, B 0.000, C 0.000 }
gfCNCPoint4[28328] = {X 120.2647, Y 41.0656, Z -6.3333, A 0.000, B 0.000, C 0.000 }
gfCNCPoint4[28329] = {X 120.4160, Y 41.1901, Z -6.3333, A 0.000, B 0.000, C 0.000 }
gfCNCPoint4[28330] = {X 120.9967, Y 41.8157, Z -6.3333, A 0.000, B 0.000, C 0.000 }
gfCNCPoint4[28331] = {X 121.4315, Y 42.5502, Z -6.3333, A 0.000, B 0.000, C 0.000 }
gfCNCPoint4[28332] = {X 121.7005, Y 43.3602, Z -6.3333, A 0.000, B 0.000, C 0.000 }
gfCNCPoint4[28333] = {X 121.7916, Y 44.2089, Z -6.3333, A 0.000, B 0.000, C 0.000 }
gfCNCPoint4[28334] = {X 121.7916, Y 45.0000, Z -6.3333, A 0.000, B 0.000, C 0.000 }
gfCNCPoint4[28335] = {X 121.6913, Y 45.8901, Z -6.3333, A 0.000, B 0.000, C 0.000 }
gfCNCPoint4[28336] = {X 121.3955, Y 46.7355, Z -6.3333, A 0.000, B 0.000, C 0.000 }
gfCNCPoint4[28337] = {X 120.9189, Y 47.4940, Z -6.3333, A 0.000, B 0.000, C 0.000 }
gfCNCPoint4[28338] = {X 120.2855, Y 48.1273, Z -6.3333, A 0.000, B 0.000, C 0.000 }
gfCNCPoint4[28339] = {X 119.5271, Y 48.6039, Z -6.3333, A 0.000, B 0.000, C 0.000 }
gfCNCPoint4[28340] = {X 118.6817, Y 48.8997, Z -6.3333, A 0.000, B 0.000, C 0.000 }
gfCNCPoint4[28341] = {X 117.7916, Y 49.0000, Z -6.3333, A 0.000, B 0.000, C 0.000 }
gfCNCPoint4[28342] = {X 111.9185, Y 49.0000, Z -6.3333, A 0.000, B 0.000, C 0.000 }
gfCNCPoint4[28343] = {X 111.0284, Y 48.8997, Z -6.3333, A 0.000, B 0.000, C 0.000 }
gfCNCPoint4[28344] = {X 110.1829, Y 48.6039, Z -6.3333, A 0.000, B 0.000, C 0.000 }
gfCNCPoint4[28345] = {X 109.4245, Y 48.1273, Z -6.3333, A 0.000, B 0.000, C 0.000 }
gfCNCPoint4[28346] = {X 108.7911, Y 47.4939, Z -6.3333, A 0.000, B 0.000, C 0.000 }
gfCNCPoint4[28347] = {X 108.3146, Y 46.7355, Z -6.3333, A 0.000, B 0.000, C 0.000 }
gfCNCPoint4[28348] = {X 108.0188, Y 45.8901, Z -6.3333, A 0.000, B 0.000, C 0.000 }
gfCNCPoint4[28349] = {X 107.9185, Y 45.0000, Z -6.3333, A 0.000, B 0.000, C 0.000 }
gfCNCPoint4[28350] = {X 107.9185, Y 44.1789, Z -6.3333, A 0.000, B 0.000, C 0.000 }
gfCNCPoint4[28351] = {X 107.9513, Y 43.6783, Z -6.3333, A 0.000, B 0.000, C 0.000 }
gfCNCPoint4[28352] = {X 108.0491, Y 43.1863, Z -6.3333, A 0.000, B 0.000, C 0.000 }
gfCNCPoint4[28353] = {X 108.2043, Y 42.7259, Z -6.3333, A 0.000, B 0.000, C 0.000 }
gfCNCPoint4[28354] = {X 108.4164, Y 42.2888, Z -6.3333, A 0.000, B 0.000, C 0.000 }
gfCNCPoint4[28355] = {X 108.4425, Y 42.2434, Z -6.3333, A 0.000, B 0.000, C 0.000 }
gfCNCPoint4[28356] = {X 108.4692, Y 42.1984, Z -6.3333, A 0.000, B 0.000, C 0.000 }
gfCNCPoint4[28357] = {X 108.9149, Y 41.5646, Z -6.3333, A 0.000, B 0.000, C 0.000 }
gfCNCPoint4[28358] = {X 109.4453, Y 40.9999, Z -6.3333, A 0.000, B 0.000, C 0.000 }
gfCNCPoint4[28359] = {X 109.4451, Y 38.9229, Z -6.3333, A 0.000, B 0.000, C 0.000 }
gfCNCPoint4[28360] = {X 108.9328, Y 38.9229, Z -6.3333, A 0.000, B 0.000, C 0.000 }
gfCNCPoint4[28361] = {X 105.8164, Y 46.5384, Z -6.3333, A 0.000, B 0.000, C 0.000 }
gfCNCPoint4[28362] = {X 105.3339, Y 47.3869, Z -6.3333, A 0.000, B 0.000, C 0.000 }
gfCNCPoint4[28363] = {X 104.6602, Y 48.0932, Z -6.3333, A 0.000, B 0.000, C 0.000 }
gfCNCPoint4[28364] = {X 103.8355, Y 48.6154, Z -6.3333, A 0.000, B 0.000, C 0.000 }
gfCNCPoint4[28365] = {X 102.9580, Y 48.9121, Z -6.3333, A 0.000, B 0.000, C 0.000 }
gfCNCPoint4[28366] = {X 102.0357, Y 48.9990, Z -6.3333, A 0.000, B 0.000, C 0.000 }
gfCNCPoint4[28367] = {X 101.1182, Y 48.8715, Z -6.3333, A 0.000, B 0.000, C 0.000 }
gfCNCPoint4[28368] = {X 100.2546, Y 48.5362, Z -6.3333, A 0.000, B 0.000, C 0.000 }
gfCNCPoint4[28369] = {X 99.4912, Y 48.0114, Z -6.3333, A 0.000, B 0.000, C 0.000 }
gfCNCPoint4[28370] = {X 98.8691, Y 47.3250, Z -6.3333, A 0.000, B 0.000, C 0.000 }
gfCNCPoint4[28371] = {X 98.4216, Y 46.5139, Z -6.3333, A 0.000, B 0.000, C 0.000 }
gfCNCPoint4[28372] = {X 94.8155, Y 37.6945, Z -6.3333, A 0.000, B 0.000, C 0.000 }
gfCNCPoint4[28373] = {X 94.8116, Y 38.2306, Z -6.3333, A 0.000, B 0.000, C 0.000 }
gfCNCPoint4[28374] = {X 94.8117, Y 41.0548, Z -6.3333, A 0.000, B 0.000, C 0.000 }
gfCNCPoint4[28375] = {X 95.3640, Y 41.5910, Z -6.3333, A 0.000, B 0.000, C 0.000 }
gfCNCPoint4[28376] = {X 95.8057, Y 42.2213, Z -6.3333, A 0.000, B 0.000, C 0.000 }
gfCNCPoint4[28377] = {X 96.0351, Y 42.6932, Z -6.3333, A 0.000, B 0.000, C 0.000 }
gfCNCPoint4[28378] = {X 96.2020, Y 43.1905, Z -6.3333, A 0.000, B 0.000, C 0.000 }
gfCNCPoint4[28379] = {X 96.3025, Y 43.6954, Z -6.3333, A 0.000, B 0.000, C 0.000 }
gfCNCPoint4[28380] = {X 96.3385, Y 44.2089, Z -6.3333, A 0.000, B 0.000, C 0.000 }
gfCNCPoint4[28381] = {X 96.3384, Y 45.0384, Z -6.3333, A 0.000, B 0.000, C 0.000 }
gfCNCPoint4[28382] = {X 96.2308, Y 45.9222, Z -6.3333, A 0.000, B 0.000, C 0.000 }
gfCNCPoint4[28383] = {X 95.9304, Y 46.7602, Z -6.3333, A 0.000, B 0.000, C 0.000 }
gfCNCPoint4[28384] = {X 95.4521, Y 47.5111, Z -6.3333, A 0.000, B 0.000, C 0.000 }
gfCNCPoint4[28385] = {X 94.8196, Y 48.1376, Z -6.3333, A 0.000, B 0.000, C 0.000 }
gfCNCPoint4[28386] = {X 94.0642, Y 48.6086, Z -6.3333, A 0.000, B 0.000, C 0.000 }
gfCNCPoint4[28387] = {X 93.2233, Y 48.9009, Z -6.3333, A 0.000, B 0.000, C 0.000 }
gfCNCPoint4[28388] = {X 92.3385, Y 49.0000, Z -6.3333, A 0.000, B 0.000, C 0.000 }
gfCNCPoint4[28389] = {X 85.8951, Y 49.0000, Z -6.3333, A 0.000, B 0.000, C 0.000 }
gfCNCPoint4[28390] = {X 85.0050, Y 48.8997, Z -6.3333, A 0.000, B 0.000, C 0.000 }
gfCNCPoint4[28391] = {X 84.1595, Y 48.6039, Z -6.3333, A 0.000, B 0.000, C 0.000 }
gfCNCPoint4[28392] = {X 83.4011, Y 48.1273, Z -6.3333, A 0.000, B 0.000, C 0.000 }
gfCNCPoint4[28393] = {X 82.7677, Y 47.4939, Z -6.3333, A 0.000, B 0.000, C 0.000 }
gfCNCPoint4[28394] = {X 82.2912, Y 46.7355, Z -6.3333, A 0.000, B 0.000, C 0.000 }
gfCNCPoint4[28395] = {X 81.9954, Y 45.8901, Z -6.3333, A 0.000, B 0.000, C 0.000 }
gfCNCPoint4[28396] = {X 81.8951, Y 45.0000, Z -6.3333, A 0.000, B 0.000, C 0.000 }
gfCNCPoint4[28397] = {X 81.8951, Y 44.2089, Z -6.3333, A 0.000, B 0.000, C 0.000 }
gfCNCPoint4[28398] = {X 82.0003, Y 43.3121, Z -6.3333, A 0.000, B 0.000, C 0.000 }
gfCNCPoint4[28399] = {X 82.3014, Y 42.4608, Z -6.3333, A 0.000, B 0.000, C 0.000 }
gfCNCPoint4[28400] = {X 82.7833, Y 41.6973, Z -6.3333, A 0.000, B 0.000, C 0.000 }
gfCNCPoint4[28401] = {X 83.4222, Y 41.0593, Z -6.3333, A 0.000, B 0.000, C 0.000 }
gfCNCPoint4[28402] = {X 83.4220, Y 28.5912, Z -6.3333, A 0.000, B 0.000, C 0.000 }
gfCNCPoint4[28403] = {X 79.3420, Y 28.5912, Z -6.3333, A 0.000, B 0.000, C 0.000 }
gfCNCPoint4[28404] = {X 79.3420, Y 28.5912, Z -3.3333, A 0.000, B 0.000, C 0.000 }
gfCNCPoint4[28405] = {X 79.3420, Y 28.5912, Z 11.0000, A 0.000, B 0.000, C 0.000 }
gfCNCPoint4[28406] = {X 136.1636, Y 30.3968, Z 11.0000, A 0.000, B 0.000, C 0.000 }
gfCNCPoint4[28407] = {X 136.1636, Y 30.3968, Z -3.3333, A 0.000, B 0.000, C 0.000 }
gfCNCPoint4[28408] = {X 136.1636, Y 30.3968, Z -6.3333, A 0.000, B 0.000, C 0.000 }
gfCNCPoint4[28409] = {X 140.2436, Y 30.3968, Z -6.3333, A 0.000, B 0.000, C 0.000 }
gfCNCPoint4[28410] = {X 140.2436, Y 19.8780, Z -6.3333, A 0.000, B 0.000, C 0.000 }
gfCNCPoint4[28411] = {X 137.4236, Y 19.8776, Z -6.3333, A 0.000, B 0.000, C 0.000 }
gfCNCPoint4[28412] = {X 136.8912, Y 20.5221, Z -6.3333, A 0.000, B 0.000, C 0.000 }
gfCNCPoint4[28413] = {X 136.2446, Y 21.0520, Z -6.3333, A 0.000, B 0.000, C 0.000 }
gfCNCPoint4[28414] = {X 135.5081, Y 21.4475, Z -6.3333, A 0.000, B 0.000, C 0.000 }
gfCNCPoint4[28415] = {X 134.7092, Y 21.6937, Z -6.3333, A 0.000, B 0.000, C 0.000 }
gfCNCPoint4[28416] = {X 133.8778, Y 21.7814, Z -6.3333, A 0.000, B 0.000, C 0.000 }
gfCNCPoint4[28417] = {X 133.2006, Y 21.7815, Z -6.3333, A 0.000, B 0.000, C 0.000 }
gfCNCPoint4[28418] = {X 132.2394, Y 21.6732, Z -6.3333, A 0.000, B 0.000, C 0.000 }
gfCNCPoint4[28419] = {X 131.3263, Y 21.3537, Z -6.3333, A 0.000, B 0.000, C 0.000 }
gfCNCPoint4[28420] = {X 130.5072, Y 20.8390, Z -6.3333, A 0.000, B 0.000, C 0.000 }
gfCNCPoint4[28421] = {X 129.8231, Y 20.1550, Z -6.3333, A 0.000, B 0.000, C 0.000 }
gfCNCPoint4[28422] = {X 129.3085, Y 19.3359, Z -6.3333, A 0.000, B 0.000, C 0.000 }
gfCNCPoint4[28423] = {X 128.9890, Y 18.4228, Z -6.3333, A 0.000, B 0.000, C 0.000 }
gfCNCPoint4[28424] = {X 128.8806, Y 17.4615, Z -6.3333, A 0.000, B 0.000, C 0.000 }
gfCNCPoint4[28425] = {X 128.8806, Y 10.4835, Z -6.3333, A 0.000, B 0.000, C 0.000 }
gfCNCPoint4[28426] = {X 128.9874, Y 9.5289, Z -6.3333, A 0.000, B 0.000, C 0.000 }
gfCNCPoint4[28427] = {X 129.3026, Y 8.6214, Z -6.3333, A 0.000, B 0.000, C 0.000 }
gfCNCPoint4[28428] = {X 129.8104, Y 7.8061, Z -6.3333, A 0.000, B 0.000, C 0.000 }
gfCNCPoint4[28429] = {X 130.4859, Y 7.1231, Z -6.3333, A 0.000, B 0.000, C 0.000 }
gfCNCPoint4[28430] = {X 131.2956, Y 6.6063, Z -6.3333, A 0.000, B 0.000, C 0.000 }
gfCNCPoint4[28431] = {X 132.1995, Y 6.2811, Z -6.3333, A 0.000, B 0.000, C 0.000 }
gfCNCPoint4[28432] = {X 133.1529, Y 6.1638, Z -6.3333, A 0.000, B 0.000, C 0.000 }
gfCNCPoint4[28433] = {X 133.8866, Y 6.1637, Z -6.3333, A 0.000, B 0.000, C 0.000 }
gfCNCPoint4[28434] = {X 134.7109, Y 6.2517, Z -6.3333, A 0.000, B 0.000, C 0.000 }
gfCNCPoint4[28435] = {X 135.5032, Y 6.4956, Z -6.3333, A 0.000, B 0.000, C 0.000 }
gfCNCPoint4[28436] = {X 136.2344, Y 6.8862, Z -6.3333, A 0.000, B 0.000, C 0.000 }
gfCNCPoint4[28437] = {X 136.8774, Y 7.4094, Z -6.3333, A 0.000, B 0.000, C 0.000 }
gfCNCPoint4[28438] = {X 137.4087, Y 8.0457, Z -6.3333, A 0.000, B 0.000, C 0.000 }
gfCNCPoint4[28439] = {X 155.1131, Y 8.0470, Z -6.3333, A 0.000, B 0.000, C 0.000 }
gfCNCPoint4[28440] = {X 155.6451, Y 7.4095, Z -6.3333, A 0.000, B 0.000, C 0.000 }
gfCNCPoint4[28441] = {X 156.2893, Y 6.8856, Z -6.3333, A 0.000, B 0.000, C 0.000 }
gfCNCPoint4[28442] = {X 157.0218, Y 6.4946, Z -6.3333, A 0.000, B 0.000, C 0.000 }
gfCNCPoint4[28443] = {X 157.8155, Y 6.2510, Z -6.3333, A 0.000, B 0.000, C 0.000 }
gfCNCPoint4[28444] = {X 158.6412, Y 6.1637, Z -6.3333, A 0.000, B 0.000, C 0.000 }
gfCNCPoint4[28445] = {X 159.3781, Y 6.1639, Z -6.3333, A 0.000, B 0.000, C 0.000 }
gfCNCPoint4[28446] = {X 160.3301, Y 6.2828, Z -6.3333, A 0.000, B 0.000, C 0.000 }
gfCNCPoint4[28447] = {X 161.2324, Y 6.6088, Z -6.3333, A 0.000, B 0.000, C 0.000 }
gfCNCPoint4[28448] = {X 162.0405, Y 7.1260, Z -6.3333, A 0.000, B 0.000, C 0.000 }
gfCNCPoint4[28449] = {X 162.7145, Y 7.8088, Z -6.3333, A 0.000, B 0.000, C 0.000 }
gfCNCPoint4[28450] = {X 163.2212, Y 8.6236, Z -6.3333, A 0.000, B 0.000, C 0.000 }
gfCNCPoint4[28451] = {X 163.5355, Y 9.5300, Z -6.3333, A 0.000, B 0.000, C 0.000 }
gfCNCPoint4[28452] = {X 163.6421, Y 10.4835, Z -6.3333, A 0.000, B 0.000, C 0.000 }
gfCNCPoint4[28453] = {X 163.6421, Y 17.4615, Z -6.3333, A 0.000, B 0.000, C 0.000 }
gfCNCPoint4[28454] = {X 163.5355, Y 18.4152, Z -6.3333, A 0.000, B 0.000, C 0.000 }
gfCNCPoint4[28455] = {X 163.2211, Y 19.3218, Z -6.3333, A 0.000, B 0.000, C 0.000 }
gfCNCPoint4[28456] = {X 162.7142, Y 20.1366, Z -6.3333, A 0.000, B 0.000, C 0.000 }
gfCNCPoint4[28457] = {X 162.0400, Y 20.8194, Z -6.3333, A 0.000, B 0.000, C 0.000 }
gfCNCPoint4[28458] = {X 161.2318, Y 21.3365, Z -6.3333, A 0.000, B 0.000, C 0.000 }
gfCNCPoint4[28459] = {X 160.3292, Y 21.6625, Z -6.3333, A 0.000, B 0.000, C 0.000 }
gfCNCPoint4[28460] = {X 159.3770, Y 21.7812, Z -6.3333, A 0.000, B 0.000, C 0.000 }
gfCNCPoint4[28461] = {X 158.6793, Y 21.7815, Z -6.3333, A 0.000, B 0.000, C 0.000 }
gfCNCPoint4[28462] = {X 157.8409, Y 21.6969, Z -6.3333, A 0.000, B 0.000, C 0.000 }
gfCNCPoint4[28463] = {X 157.0346, Y 21.4522, Z -6.3333, A 0.000, B 0.000, C 0.000 }
gfCNCPoint4[28464] = {X 156.2905, Y 21.0567, Z -6.3333, A 0.000, B 0.000, C 0.000 }
gfCNCPoint4[28465] = {X 155.6366, Y 20.5252, Z -6.3333, A 0.000, B 0.000, C 0.000 }
gfCNCPoint4[28466] = {X 155.0974, Y 19.8776, Z -6.3333, A 0.000, B 0.000, C 0.000 }
gfCNCPoint4[28467] = {X 152.2769, Y 19.8786, Z -6.3333, A 0.000, B 0.000, C 0.000 }
gfCNCPoint4[28468] = {X 152.2758, Y 40.8742, Z -6.3333, A 0.000, B 0.000, C 0.000 }
gfCNCPoint4[28469] = {X 152.7408, Y 41.3749, Z -6.3333, A 0.000, B 0.000, C 0.000 }
gfCNCPoint4[28470] = {X 152.8364, Y 41.4887, Z -6.3333, A 0.000, B 0.000, C 0.000 }
gfCNCPoint4[28471] = {X 153.3620, Y 42.3140, Z -6.3333, A 0.000, B 0.000, C 0.000 }
gfCNCPoint4[28472] = {X 153.6898, Y 43.2359, Z -6.3333, A 0.000, B 0.000, C 0.000 }
gfCNCPoint4[28473] = {X 153.8031, Y 44.2078, Z -6.3333, A 0.000, B 0.000, C 0.000 }
gfCNCPoint4[28474] = {X 153.8029, Y 45.0415, Z -6.3333, A 0.000, B 0.000, C 0.000 }
gfCNCPoint4[28475] = {X 153.6867, Y 45.9960, Z -6.3333, A 0.000, B 0.000, C 0.000 }
gfCNCPoint4[28476] = {X 153.3623, Y 46.9011, Z -6.3333, A 0.000, B 0.000, C 0.000 }
gfCNCPoint4[28477] = {X 152.8458, Y 47.7120, Z -6.3333, A 0.000, B 0.000, C 0.000 }
gfCNCPoint4[28478] = {X 152.1626, Y 48.3886, Z -6.3333, A 0.000, B 0.000, C 0.000 }
gfCNCPoint4[28479] = {X 151.3468, Y 48.8973, Z -6.3333, A 0.000, B 0.000, C 0.000 }
gfCNCPoint4[28480] = {X 150.4386, Y 49.2130, Z -6.3333, A 0.000, B 0.000, C 0.000 }
gfCNCPoint4[28481] = {X 149.4831, Y 49.3200, Z -6.3333, A 0.000, B 0.000, C 0.000 }
gfCNCPoint4[28482] = {X 143.0396, Y 49.3200, Z -6.3333, A 0.000, B 0.000, C 0.000 }
gfCNCPoint4[28483] = {X 142.0831, Y 49.2128, Z -6.3333, A 0.000, B 0.000, C 0.000 }
gfCNCPoint4[28484] = {X 141.1741, Y 48.8964, Z -6.3333, A 0.000, B 0.000, C 0.000 }
gfCNCPoint4[28485] = {X 140.3576, Y 48.3866, Z -6.3333, A 0.000, B 0.000, C 0.000 }
gfCNCPoint4[28486] = {X 139.6743, Y 47.7087, Z -6.3333, A 0.000, B 0.000, C 0.000 }
gfCNCPoint4[28487] = {X 139.1581, Y 46.8964, Z -6.3333, A 0.000, B 0.000, C 0.000 }
gfCNCPoint4[28488] = {X 138.8346, Y 45.9899, Z -6.3333, A 0.000, B 0.000, C 0.000 }
gfCNCPoint4[28489] = {X 138.7198, Y 45.0342, Z -6.3333, A 0.000, B 0.000, C 0.000 }
gfCNCPoint4[28490] = {X 138.7200, Y 44.1494, Z -6.3333, A 0.000, B 0.000, C 0.000 }
gfCNCPoint4[28491] = {X 138.8305, Y 43.2364, Z -6.3333, A 0.000, B 0.000, C 0.000 }
gfCNCPoint4[28492] = {X 139.1317, Y 42.3675, Z -6.3333, A 0.000, B 0.000, C 0.000 }
gfCNCPoint4[28493] = {X 139.6099, Y 41.5821, Z -6.3333, A 0.000, B 0.000, C 0.000 }
gfCNCPoint4[28494] = {X 140.2436, Y 40.9157, Z -6.3333, A 0.000, B 0.000, C 0.000 }
gfCNCPoint4[28495] = {X 140.2436, Y 30.3968, Z -6.3333, A 0.000, B 0.000, C 0.000 }
gfCNCPoint4[28496] = {X 136.2436, Y 30.3968, Z -6.3333, A 0.000, B 0.000, C 0.000 }
gfCNCPoint4[28497] = {X 140.3236, Y 30.3968, Z -6.3333, A 0.000, B 0.000, C 0.000 }
gfCNCPoint4[28498] = {X 140.3236, Y 19.7980, Z -6.3333, A 0.000, B 0.000, C 0.000 }
gfCNCPoint4[28499] = {X 137.3794, Y 19.7975, Z -6.3333, A 0.000, B 0.000, C 0.000 }
gfCNCPoint4[28500] = {X 137.3565, Y 19.8338, Z -6.3333, A 0.000, B 0.000, C 0.000 }
gfCNCPoint4[28501] = {X 136.8340, Y 20.4661, Z -6.3333, A 0.000, B 0.000, C 0.000 }
gfCNCPoint4[28502] = {X 136.1995, Y 20.9859, Z -6.3333, A 0.000, B 0.000, C 0.000 }
gfCNCPoint4[28503] = {X 135.4768, Y 21.3738, Z -6.3333, A 0.000, B 0.000, C 0.000 }
gfCNCPoint4[28504] = {X 134.6929, Y 21.6153, Z -6.3333, A 0.000, B 0.000, C 0.000 }
gfCNCPoint4[28505] = {X 133.8772, Y 21.7014, Z -6.3333, A 0.000, B 0.000, C 0.000 }
gfCNCPoint4[28506] = {X 133.2006, Y 21.7015, Z -6.3333, A 0.000, B 0.000, C 0.000 }
gfCNCPoint4[28507] = {X 132.2572, Y 21.5952, Z -6.3333, A 0.000, B 0.000, C 0.000 }
gfCNCPoint4[28508] = {X 131.3610, Y 21.2816, Z -6.3333, A 0.000, B 0.000, C 0.000 }
gfCNCPoint4[28509] = {X 130.5570, Y 20.7765, Z -6.3333, A 0.000, B 0.000, C 0.000 }
gfCNCPoint4[28510] = {X 129.8857, Y 20.1051, Z -6.3333, A 0.000, B 0.000, C 0.000 }
gfCNCPoint4[28511] = {X 129.3805, Y 19.3012, Z -6.3333, A 0.000, B 0.000, C 0.000 }
gfCNCPoint4[28512] = {X 129.0669, Y 18.4050, Z -6.3333, A 0.000, B 0.000, C 0.000 }
gfCNCPoint4[28513] = {X 128.9606, Y 17.4615, Z -6.3333, A 0.000, B 0.000, C 0.000 }
gfCNCPoint4[28514] = {X 128.9606, Y 10.4835, Z -6.3333, A 0.000, B 0.000, C 0.000 }
gfCNCPoint4[28515] = {X 129.0655, Y 9.5466, Z -6.3333, A 0.000, B 0.000, C 0.000 }
gfCNCPoint4[28516] = {X 129.3747, Y 8.6559, Z -6.3333, A 0.000, B 0.000, C 0.000 }
gfCNCPoint4[28517] = {X 129.8732, Y 7.8557, Z -6.3333, A 0.000, B 0.000, C 0.000 }
gfCNCPoint4[28518] = {X 130.5362, Y 7.1853, Z -6.3333, A 0.000, B 0.000, C 0.000 }
gfCNCPoint4[28519] = {X 131.3309, Y 6.6781, Z -6.3333, A 0.000, B 0.000, C 0.000 }
gfCNCPoint4[28520] = {X 132.2180, Y 6.3589, Z -6.3333, A 0.000, B 0.000, C 0.000 }
gfCNCPoint4[28521] = {X 133.1538, Y 6.2438, Z -6.3333, A 0.000, B 0.000, C 0.000 }
gfCNCPoint4[28522] = {X 133.8858, Y 6.2437, Z -6.3333, A 0.000, B 0.000, C 0.000 }
gfCNCPoint4[28523] = {X 134.7031, Y 6.3318, Z -6.3333, A 0.000, B 0.000, C 0.000 }
gfCNCPoint4[28524] = {X 135.4880, Y 6.5759, Z -6.3333, A 0.000, B 0.000, C 0.000 }
gfCNCPoint4[28525] = {X 136.2110, Y 6.9669, Z -6.3333, A 0.000, B 0.000, C 0.000 }
gfCNCPoint4[28526] = {X 136.8451, Y 7.4900, Z -6.3333, A 0.000, B 0.000, C 0.000 }
gfCNCPoint4[28527] = {X 137.3663, Y 8.1257, Z -6.3333, A 0.000, B 0.000, C 0.000 }
gfCNCPoint4[28528] = {X 155.1556, Y 8.1270, Z -6.3333, A 0.000, B 0.000, C 0.000 }
gfCNCPoint4[28529] = {X 155.6775, Y 7.4902, Z -6.3333, A 0.000, B 0.000, C 0.000 }
gfCNCPoint4[28530] = {X 156.3126, Y 6.9663, Z -6.3333, A 0.000, B 0.000, C 0.000 }
gfCNCPoint4[28531] = {X 157.0369, Y 6.5750, Z -6.3333, A 0.000, B 0.000, C 0.000 }
gfCNCPoint4[28532] = {X 157.8233, Y 6.3311, Z -6.3333, A 0.000, B 0.000, C 0.000 }
gfCNCPoint4[28533] = {X 158.6420, Y 6.2437, Z -6.3333, A 0.000, B 0.000, C 0.000 }
gfCNCPoint4[28534] = {X 159.3770, Y 6.2439, Z -6.3333, A 0.000, B 0.000, C 0.000 }
gfCNCPoint4[28535] = {X 160.3114, Y 6.3606, Z -6.3333, A 0.000, B 0.000, C 0.000 }
gfCNCPoint4[28536] = {X 161.1970, Y 6.6806, Z -6.3333, A 0.000, B 0.000, C 0.000 }
gfCNCPoint4[28537] = {X 161.9902, Y 7.1882, Z -6.3333, A 0.000, B 0.000, C 0.000 }
gfCNCPoint4[28538] = {X 162.6517, Y 7.8584, Z -6.3333, A 0.000, B 0.000, C 0.000 }
gfCNCPoint4[28539] = {X 163.1490, Y 8.6580, Z -6.3333, A 0.000, B 0.000, C 0.000 }
gfCNCPoint4[28540] = {X 163.4575, Y 9.5477, Z -6.3333, A 0.000, B 0.000, C 0.000 }
gfCNCPoint4[28541] = {X 163.5621, Y 10.4835, Z -6.3333, A 0.000, B 0.000, C 0.000 }
gfCNCPoint4[28542] = {X 163.5621, Y 17.4615, Z -6.3333, A 0.000, B 0.000, C 0.000 }
gfCNCPoint4[28543] = {X 163.4575, Y 18.3975, Z -6.3333, A 0.000, B 0.000, C 0.000 }
gfCNCPoint4[28544] = {X 163.1489, Y 19.2873, Z -6.3333, A 0.000, B 0.000, C 0.000 }
gfCNCPoint4[28545] = {X 162.6514, Y 20.0870, Z -6.3333, A 0.000, B 0.000, C 0.000 }
gfCNCPoint4[28546] = {X 161.9897, Y 20.7572, Z -6.3333, A 0.000, B 0.000, C 0.000 }
gfCNCPoint4[28547] = {X 161.1964, Y 21.2648, Z -6.3333, A 0.000, B 0.000, C 0.000 }
gfCNCPoint4[28548] = {X 160.3106, Y 21.5847, Z -6.3333, A 0.000, B 0.000, C 0.000 }
gfCNCPoint4[28549] = {X 159.3760, Y 21.7012, Z -6.3333, A 0.000, B 0.000, C 0.000 }
gfCNCPoint4[28550] = {X 158.6796, Y 21.7015, Z -6.3333, A 0.000, B 0.000, C 0.000 }
gfCNCPoint4[28551] = {X 157.8484, Y 21.6168, Z -6.3333, A 0.000, B 0.000, C 0.000 }
gfCNCPoint4[28552] = {X 157.0495, Y 21.3718, Z -6.3333, A 0.000, B 0.000, C 0.000 }
gfCNCPoint4[28553] = {X 156.3136, Y 20.9759, Z -6.3333, A 0.000, B 0.000, C 0.000 }
gfCNCPoint4[28554] = {X 155.6689, Y 20.4444, Z -6.3333, A 0.000, B 0.000, C 0.000 }
gfCNCPoint4[28555] = {X 155.1399, Y 19.7976, Z -6.3333, A 0.000, B 0.000, C 0.000 }
gfCNCPoint4[28556] = {X 152.1969, Y 19.7986, Z -6.3333, A 0.000, B 0.000, C 0.000 }
gfCNCPoint4[28557] = {X 152.1958, Y 40.9056, Z -6.3333, A 0.000, B 0.000, C 0.000 }
gfCNCPoint4[28558] = {X 152.6808, Y 41.4279, Z -6.3333, A 0.000, B 0.000, C 0.000 }
gfCNCPoint4[28559] = {X 152.7747, Y 41.5396, Z -6.3333, A 0.000, B 0.000, C 0.000 }
gfCNCPoint4[28560] = {X 153.2904, Y 42.3496, Z -6.3333, A 0.000, B 0.000, C 0.000 }
gfCNCPoint4[28561] = {X 153.6119, Y 43.2543, Z -6.3333, A 0.000, B 0.000, C 0.000 }
gfCNCPoint4[28562] = {X 153.7231, Y 44.2081, Z -6.3333, A 0.000, B 0.000, C 0.000 }
gfCNCPoint4[28563] = {X 153.7229, Y 45.0408, Z -6.3333, A 0.000, B 0.000, C 0.000 }
gfCNCPoint4[28564] = {X 153.6089, Y 45.9775, Z -6.3333, A 0.000, B 0.000, C 0.000 }
gfCNCPoint4[28565] = {X 153.2905, Y 46.8659, Z -6.3333, A 0.000, B 0.000, C 0.000 }
gfCNCPoint4[28566] = {X 152.7835, Y 47.6618, Z -6.3333, A 0.000, B 0.000, C 0.000 }
gfCNCPoint4[28567] = {X 152.1130, Y 48.3258, Z -6.3333, A 0.000, B 0.000, C 0.000 }
gfCNCPoint4[28568] = {X 151.3123, Y 48.8251, Z -6.3333, A 0.000, B 0.000, C 0.000 }
gfCNCPoint4[28569] = {X 150.4209, Y 49.1350, Z -6.3333, A 0.000, B 0.000, C 0.000 }
gfCNCPoint4[28570] = {X 149.4831, Y 49.2400, Z -6.3333, A 0.000, B 0.000, C 0.000 }
gfCNCPoint4[28571] = {X 143.0396, Y 49.2400, Z -6.3333, A 0.000, B 0.000, C 0.000 }
gfCNCPoint4[28572] = {X 142.1008, Y 49.1348, Z -6.3333, A 0.000, B 0.000, C 0.000 }
gfCNCPoint4[28573] = {X 141.2086, Y 48.8243, Z -6.3333, A 0.000, B 0.000, C 0.000 }
gfCNCPoint4[28574] = {X 140.4073, Y 48.3239, Z -6.3333, A 0.000, B 0.000, C 0.000 }
gfCNCPoint4[28575] = {X 139.7367, Y 47.6586, Z -6.3333, A 0.000, B 0.000, C 0.000 }
gfCNCPoint4[28576] = {X 139.2300, Y 46.8612, Z -6.3333, A 0.000, B 0.000, C 0.000 }
gfCNCPoint4[28577] = {X 138.9124, Y 45.9715, Z -6.3333, A 0.000, B 0.000, C 0.000 }
gfCNCPoint4[28578] = {X 138.7998, Y 45.0336, Z -6.3333, A 0.000, B 0.000, C 0.000 }
gfCNCPoint4[28579] = {X 138.8000, Y 44.1505, Z -6.3333, A 0.000, B 0.000, C 0.000 }
gfCNCPoint4[28580] = {X 138.9105, Y 43.2454, Z -6.3333, A 0.000, B 0.000, C 0.000 }
gfCNCPoint4[28581] = {X 139.2119, Y 42.3850, Z -6.3333, A 0.000, B 0.000, C 0.000 }
gfCNCPoint4[28582] = {X 139.6903, Y 41.6088, Z -6.3333, A 0.000, B 0.000, C 0.000 }
gfCNCPoint4[28583] = {X 140.3236, Y 40.9529, Z -6.3333, A 0.000, B 0.000, C 0.000 }
gfCNCPoint4[28584] = {X 140.3236, Y 30.3968, Z -6.3333, A 0.000, B 0.000, C 0.000 }
gfCNCPoint4[28585] = {X 136.3236, Y 30.3968, Z -6.3333, A 0.000, B 0.000, C 0.000 }
gfCNCPoint4[28586] = {X 140.4036, Y 30.3968, Z -6.3333, A 0.000, B 0.000, C 0.000 }
gfCNCPoint4[28587] = {X 140.4036, Y 19.7180, Z -6.3333, A 0.000, B 0.000, C 0.000 }
gfCNCPoint4[28588] = {X 137.3352, Y 19.7175, Z -6.3333, A 0.000, B 0.000, C 0.000 }
gfCNCPoint4[28589] = {X 137.2895, Y 19.7901, Z -6.3333, A 0.000, B 0.000, C 0.000 }
gfCNCPoint4[28590] = {X 136.7768, Y 20.4101, Z -6.3333, A 0.000, B 0.000, C 0.000 }
gfCNCPoint4[28591] = {X 136.1544, Y 20.9199, Z -6.3333, A 0.000, B 0.000, C 0.000 }
gfCNCPoint4[28592] = {X 135.4455, Y 21.3002, Z -6.3333, A 0.000, B 0.000, C 0.000 }
gfCNCPoint4[28593] = {X 134.6766, Y 21.5370, Z -6.3333, A 0.000, B 0.000, C 0.000 }
gfCNCPoint4[28594] = {X 133.8765, Y 21.6214, Z -6.3333, A 0.000, B 0.000, C 0.000 }
gfCNCPoint4[28595] = {X 133.2006, Y 21.6215, Z -6.3333, A 0.000, B 0.000, C 0.000 }
gfCNCPoint4[28596] = {X 132.2750, Y 21.5172, Z -6.3333, A 0.000, B 0.000, C 0.000 }
gfCNCPoint4[28597] = {X 131.3957, Y 21.2096, Z -6.3333, A 0.000, B 0.000, C 0.000 }
gfCNCPoint4[28598] = {X 130.6069, Y 20.7140, Z -6.3333, A 0.000, B 0.000, C 0.000 }
gfCNCPoint4[28599] = {X 129.9482, Y 20.0553, Z -6.3333, A 0.000, B 0.000, C 0.000 }
gfCNCPoint4[28600] = {X 129.4526, Y 19.2665, Z -6.3333, A 0.000, B 0.000, C 0.000 }
gfCNCPoint4[28601] = {X 129.1449, Y 18.3872, Z -6.3333, A 0.000, B 0.000, C 0.000 }
gfCNCPoint4[28602] = {X 129.0406, Y 17.4615, Z -6.3333, A 0.000, B 0.000, C 0.000 }
gfCNCPoint4[28603] = {X 129.0406, Y 10.4835, Z -6.3333, A 0.000, B 0.000, C 0.000 }
gfCNCPoint4[28604] = {X 129.1435, Y 9.5642, Z -6.3333, A 0.000, B 0.000, C 0.000 }
gfCNCPoint4[28605] = {X 129.4469, Y 8.6904, Z -6.3333, A 0.000, B 0.000, C 0.000 }
gfCNCPoint4[28606] = {X 129.9360, Y 7.9052, Z -6.3333, A 0.000, B 0.000, C 0.000 }
gfCNCPoint4[28607] = {X 130.5864, Y 7.2475, Z -6.3333, A 0.000, B 0.000, C 0.000 }
gfCNCPoint4[28608] = {X 131.3661, Y 6.7499, Z -6.3333, A 0.000, B 0.000, C 0.000 }
gfCNCPoint4[28609] = {X 132.2366, Y 6.4368, Z -6.3333, A 0.000, B 0.000, C 0.000 }
gfCNCPoint4[28610] = {X 133.1547, Y 6.3238, Z -6.3333, A 0.000, B 0.000, C 0.000 }
gfCNCPoint4[28611] = {X 133.8850, Y 6.3237, Z -6.3333, A 0.000, B 0.000, C 0.000 }
gfCNCPoint4[28612] = {X 134.6952, Y 6.4119, Z -6.3333, A 0.000, B 0.000, C 0.000 }
gfCNCPoint4[28613] = {X 135.4726, Y 6.6563, Z -6.3333, A 0.000, B 0.000, C 0.000 }
gfCNCPoint4[28614] = {X 136.1875, Y 7.0476, Z -6.3333, A 0.000, B 0.000, C 0.000 }
gfCNCPoint4[28615] = {X 136.8124, Y 7.5707, Z -6.3333, A 0.000, B 0.000, C 0.000 }
gfCNCPoint4[28616] = {X 137.3233, Y 8.2057, Z -6.3333, A 0.000, B 0.000, C 0.000 }
gfCNCPoint4[28617] = {X 155.1986, Y 8.2070, Z -6.3333, A 0.000, B 0.000, C 0.000 }
gfCNCPoint4[28618] = {X 155.7101, Y 7.5709, Z -6.3333, A 0.000, B 0.000, C 0.000 }
gfCNCPoint4[28619] = {X 156.3361, Y 7.0470, Z -6.3333, A 0.000, B 0.000, C 0.000 }
gfCNCPoint4[28620] = {X 157.0522, Y 6.6554, Z -6.3333, A 0.000, B 0.000, C 0.000 }
gfCNCPoint4[28621] = {X 157.8311, Y 6.4111, Z -6.3333, A 0.000, B 0.000, C 0.000 }
gfCNCPoint4[28622] = {X 158.6427, Y 6.3237, Z -6.3333, A 0.000, B 0.000, C 0.000 }
gfCNCPoint4[28623] = {X 159.3760, Y 6.3239, Z -6.3333, A 0.000, B 0.000, C 0.000 }
gfCNCPoint4[28624] = {X 160.2928, Y 6.4383, Z -6.3333, A 0.000, B 0.000, C 0.000 }
gfCNCPoint4[28625] = {X 161.1617, Y 6.7524, Z -6.3333, A 0.000, B 0.000, C 0.000 }
gfCNCPoint4[28626] = {X 161.9398, Y 7.2504, Z -6.3333, A 0.000, B 0.000, C 0.000 }
gfCNCPoint4[28627] = {X 162.5889, Y 7.9079, Z -6.3333, A 0.000, B 0.000, C 0.000 }
gfCNCPoint4[28628] = {X 163.0768, Y 8.6925, Z -6.3333, A 0.000, B 0.000, C 0.000 }
gfCNCPoint4[28629] = {X 163.3795, Y 9.5653, Z -6.3333, A 0.000, B 0.000, C 0.000 }
gfCNCPoint4[28630] = {X 163.4821, Y 10.4835, Z -6.3333, A 0.000, B 0.000, C 0.000 }
gfCNCPoint4[28631] = {X 163.4821, Y 17.4615, Z -6.3333, A 0.000, B 0.000, C 0.000 }
gfCNCPoint4[28632] = {X 163.3795, Y 18.3798, Z -6.3333, A 0.000, B 0.000, C 0.000 }
gfCNCPoint4[28633] = {X 163.0767, Y 19.2527, Z -6.3333, A 0.000, B 0.000, C 0.000 }
gfCNCPoint4[28634] = {X 162.5887, Y 20.0373, Z -6.3333, A 0.000, B 0.000, C 0.000 }
gfCNCPoint4[28635] = {X 161.9396, Y 20.6948, Z -6.3333, A 0.000, B 0.000, C 0.000 }
gfCNCPoint4[28636] = {X 161.1613, Y 21.1929, Z -6.3333, A 0.000, B 0.000, C 0.000 }
gfCNCPoint4[28637] = {X 160.2923, Y 21.5068, Z -6.3333, A 0.000, B 0.000, C 0.000 }
gfCNCPoint4[28638] = {X 159.3755, Y 21.6212, Z -6.3333, A 0.000, B 0.000, C 0.000 }
gfCNCPoint4[28639] = {X 158.6799, Y 21.6215, Z -6.3333, A 0.000, B 0.000, C 0.000 }
gfCNCPoint4[28640] = {X 157.8558, Y 21.5366, Z -6.3333, A 0.000, B 0.000, C 0.000 }
gfCNCPoint4[28641] = {X 157.0646, Y 21.2913, Z -6.3333, A 0.000, B 0.000, C 0.000 }
gfCNCPoint4[28642] = {X 156.3370, Y 20.8952, Z -6.3333, A 0.000, B 0.000, C 0.000 }
gfCNCPoint4[28643] = {X 155.7015, Y 20.3637, Z -6.3333, A 0.000, B 0.000, C 0.000 }
gfCNCPoint4[28644] = {X 155.1830, Y 19.7176, Z -6.3333, A 0.000, B 0.000, C 0.000 }
gfCNCPoint4[28645] = {X 152.1169, Y 19.7187, Z -6.3333, A 0.000, B 0.000, C 0.000 }
gfCNCPoint4[28646] = {X 152.1158, Y 40.9370, Z -6.3333, A 0.000, B 0.000, C 0.000 }
gfCNCPoint4[28647] = {X 152.6209, Y 41.4808, Z -6.3333, A 0.000, B 0.000, C 0.000 }
gfCNCPoint4[28648] = {X 152.7129, Y 41.5905, Z -6.3333, A 0.000, B 0.000, C 0.000 }
gfCNCPoint4[28649] = {X 153.2187, Y 42.3851, Z -6.3333, A 0.000, B 0.000, C 0.000 }
gfCNCPoint4[28650] = {X 153.5341, Y 43.2727, Z -6.3333, A 0.000, B 0.000, C 0.000 }
gfCNCPoint4[28651] = {X 153.6431, Y 44.2083, Z -6.3333, A 0.000, B 0.000, C 0.000 }
gfCNCPoint4[28652] = {X 153.6429, Y 45.0400, Z -6.3333, A 0.000, B 0.000, C 0.000 }
gfCNCPoint4[28653] = {X 153.5310, Y 45.9591, Z -6.3333, A 0.000, B 0.000, C 0.000 }
gfCNCPoint4[28654] = {X 153.2186, Y 46.8306, Z -6.3333, A 0.000, B 0.000, C 0.000 }
gfCNCPoint4[28655] = {X 152.7212, Y 47.6115, Z -6.3333, A 0.000, B 0.000, C 0.000 }
gfCNCPoint4[28656] = {X 152.0634, Y 48.2631, Z -6.3333, A 0.000, B 0.000, C 0.000 }
gfCNCPoint4[28657] = {X 151.2778, Y 48.7530, Z -6.3333, A 0.000, B 0.000, C 0.000 }
gfCNCPoint4[28658] = {X 150.4032, Y 49.0570, Z -6.3333, A 0.000, B 0.000, C 0.000 }
gfCNCPoint4[28659] = {X 149.4831, Y 49.1600, Z -6.3333, A 0.000, B 0.000, C 0.000 }
gfCNCPoint4[28660] = {X 143.0396, Y 49.1600, Z -6.3333, A 0.000, B 0.000, C 0.000 }
gfCNCPoint4[28661] = {X 142.1185, Y 49.0567, Z -6.3333, A 0.000, B 0.000, C 0.000 }
gfCNCPoint4[28662] = {X 141.2432, Y 48.7521, Z -6.3333, A 0.000, B 0.000, C 0.000 }
gfCNCPoint4[28663] = {X 140.4570, Y 48.2612, Z -6.3333, A 0.000, B 0.000, C 0.000 }
gfCNCPoint4[28664] = {X 139.7990, Y 47.6084, Z -6.3333, A 0.000, B 0.000, C 0.000 }
gfCNCPoint4[28665] = {X 139.3019, Y 46.8261, Z -6.3333, A 0.000, B 0.000, C 0.000 }
gfCNCPoint4[28666] = {X 138.9903, Y 45.9532, Z -6.3333, A 0.000, B 0.000, C 0.000 }
gfCNCPoint4[28667] = {X 138.8798, Y 45.0329, Z -6.3333, A 0.000, B 0.000, C 0.000 }
gfCNCPoint4[28668] = {X 138.8800, Y 44.1516, Z -6.3333, A 0.000, B 0.000, C 0.000 }
gfCNCPoint4[28669] = {X 138.9906, Y 43.2545, Z -6.3333, A 0.000, B 0.000, C 0.000 }
gfCNCPoint4[28670] = {X 139.2922, Y 42.4026, Z -6.3333, A 0.000, B 0.000, C 0.000 }
gfCNCPoint4[28671] = {X 139.7708, Y 41.6358, Z -6.3333, A 0.000, B 0.000, C 0.000 }
gfCNCPoint4[28672] = {X 140.4036, Y 40.9906, Z -6.3333, A 0.000, B 0.000, C 0.000 }
gfCNCPoint4[28673] = {X 140.4036, Y 30.3968, Z -6.3333, A 0.000, B 0.000, C 0.000 }
gfCNCPoint4[28674] = {X 136.4036, Y 30.3968, Z -6.3333, A 0.000, B 0.000, C 0.000 }
gfCNCPoint4[28675] = {X 140.4836, Y 30.3968, Z -6.3333, A 0.000, B 0.000, C 0.000 }
gfCNCPoint4[28676] = {X 140.4836, Y 19.6380, Z -6.3333, A 0.000, B 0.000, C 0.000 }
gfCNCPoint4[28677] = {X 137.2910, Y 19.6375, Z -6.3333, A 0.000, B 0.000, C 0.000 }
gfCNCPoint4[28678] = {X 137.2218, Y 19.7475, Z -6.3333, A 0.000, B 0.000, C 0.000 }
gfCNCPoint4[28679] = {X 136.5756, Y 20.4907, Z -6.3333, A 0.000, B 0.000, C 0.000 }
gfCNCPoint4[28680] = {X 135.7702, Y 21.0573, Z -6.3333, A 0.000, B 0.000, C 0.000 }
gfCNCPoint4[28681] = {X 134.8524, Y 21.4145, Z -6.3333, A 0.000, B 0.000, C 0.000 }
gfCNCPoint4[28682] = {X 133.8758, Y 21.5414, Z -6.3333, A 0.000, B 0.000, C 0.000 }
gfCNCPoint4[28683] = {X 133.2006, Y 21.5415, Z -6.3333, A 0.000, B 0.000, C 0.000 }
gfCNCPoint4[28684] = {X 132.2928, Y 21.4392, Z -6.3333, A 0.000, B 0.000, C 0.000 }
gfCNCPoint4[28685] = {X 131.4304, Y 21.1375, Z -6.3333, A 0.000, B 0.000, C 0.000 }
gfCNCPoint4[28686] = {X 130.6568, Y 20.6514, Z -6.3333, A 0.000, B 0.000, C 0.000 }
gfCNCPoint4[28687] = {X 130.0108, Y 20.0054, Z -6.3333, A 0.000, B 0.000, C 0.000 }
gfCNCPoint4[28688] = {X 129.5247, Y 19.2318, Z -6.3333, A 0.000, B 0.000, C 0.000 }
gfCNCPoint4[28689] = {X 129.2229, Y 18.3694, Z -6.3333, A 0.000, B 0.000, C 0.000 }
gfCNCPoint4[28690] = {X 129.1206, Y 17.4615, Z -6.3333, A 0.000, B 0.000, C 0.000 }
gfCNCPoint4[28691] = {X 129.1206, Y 10.4835, Z -6.3333, A 0.000, B 0.000, C 0.000 }
gfCNCPoint4[28692] = {X 129.2215, Y 9.5820, Z -6.3333, A 0.000, B 0.000, C 0.000 }
gfCNCPoint4[28693] = {X 129.5191, Y 8.7250, Z -6.3333, A 0.000, B 0.000, C 0.000 }
gfCNCPoint4[28694] = {X 129.9986, Y 7.9550, Z -6.3333, A 0.000, B 0.000, C 0.000 }
gfCNCPoint4[28695] = {X 130.6365, Y 7.3099, Z -6.3333, A 0.000, B 0.000, C 0.000 }
gfCNCPoint4[28696] = {X 131.4011, Y 6.8218, Z -6.3333, A 0.000, B 0.000, C 0.000 }
gfCNCPoint4[28697] = {X 132.2547, Y 6.5147, Z -6.3333, A 0.000, B 0.000, C 0.000 }
gfCNCPoint4[28698] = {X 133.1551, Y 6.4038, Z -6.3333, A 0.000, B 0.000, C 0.000 }
gfCNCPoint4[28699] = {X 133.8841, Y 6.4037, Z -6.3333, A 0.000, B 0.000, C 0.000 }
gfCNCPoint4[28700] = {X 134.6872, Y 6.4920, Z -6.3333, A 0.000, B 0.000, C 0.000 }
gfCNCPoint4[28701] = {X 135.4571, Y 6.7367, Z -6.3333, A 0.000, B 0.000, C 0.000 }
gfCNCPoint4[28702] = {X 136.1637, Y 7.1283, Z -6.3333, A 0.000, B 0.000, C 0.000 }
gfCNCPoint4[28703] = {X 136.7793, Y 7.6515, Z -6.3333, A 0.000, B 0.000, C 0.000 }
gfCNCPoint4[28704] = {X 137.2797, Y 8.2857, Z -6.3333, A 0.000, B 0.000, C 0.000 }
gfCNCPoint4[28705] = {X 155.2421, Y 8.2870, Z -6.3333, A 0.000, B 0.000, C 0.000 }
gfCNCPoint4[28706] = {X 155.2876, Y 8.2174, Z -6.3333, A 0.000, B 0.000, C 0.000 }
gfCNCPoint4[28707] = {X 155.3344, Y 8.1488, Z -6.3333, A 0.000, B 0.000, C 0.000 }
gfCNCPoint4[28708] = {X 155.9796, Y 7.4254, Z -6.3333, A 0.000, B 0.000, C 0.000 }
gfCNCPoint4[28709] = {X 156.7771, Y 6.8747, Z -6.3333, A 0.000, B 0.000, C 0.000 }
gfCNCPoint4[28710] = {X 157.6821, Y 6.5275, Z -6.3333, A 0.000, B 0.000, C 0.000 }
gfCNCPoint4[28711] = {X 158.6434, Y 6.4037, Z -6.3333, A 0.000, B 0.000, C 0.000 }
gfCNCPoint4[28712] = {X 159.3750, Y 6.4039, Z -6.3333, A 0.000, B 0.000, C 0.000 }
gfCNCPoint4[28713] = {X 160.2741, Y 6.5161, Z -6.3333, A 0.000, B 0.000, C 0.000 }
gfCNCPoint4[28714] = {X 161.1263, Y 6.8241, Z -6.3333, A 0.000, B 0.000, C 0.000 }
gfCNCPoint4[28715] = {X 161.8895, Y 7.3126, Z -6.3333, A 0.000, B 0.000, C 0.000 }
gfCNCPoint4[28716] = {X 162.5260, Y 7.9574, Z -6.3333, A 0.000, B 0.000, C 0.000 }
gfCNCPoint4[28717] = {X 163.0046, Y 8.7269, Z -6.3333, A 0.000, B 0.000, C 0.000 }
gfCNCPoint4[28718] = {X 163.3015, Y 9.5830, Z -6.3333, A 0.000, B 0.000, C 0.000 }
gfCNCPoint4[28719] = {X 163.4021, Y 10.4835, Z -6.3333, A 0.000, B 0.000, C 0.000 }
gfCNCPoint4[28720] = {X 163.4021, Y 17.4615, Z -6.3333, A 0.000, B 0.000, C 0.000 }
gfCNCPoint4[28721] = {X 163.3015, Y 18.3621, Z -6.3333, A 0.000, B 0.000, C 0.000 }
gfCNCPoint4[28722] = {X 163.0046, Y 19.2182, Z -6.3333, A 0.000, B 0.000, C 0.000 }
gfCNCPoint4[28723] = {X 162.5260, Y 19.9876, Z -6.3333, A 0.000, B 0.000, C 0.000 }
gfCNCPoint4[28724] = {X 161.8895, Y 20.6325, Z -6.3333, A 0.000, B 0.000, C 0.000 }
gfCNCPoint4[28725] = {X 161.1263, Y 21.1209, Z -6.3333, A 0.000, B 0.000, C 0.000 }
gfCNCPoint4[28726] = {X 160.2741, Y 21.4289, Z -6.3333, A 0.000, B 0.000, C 0.000 }
gfCNCPoint4[28727] = {X 159.3750, Y 21.5412, Z -6.3333, A 0.000, B 0.000, C 0.000 }
gfCNCPoint4[28728] = {X 158.6802, Y 21.5415, Z -6.3333, A 0.000, B 0.000, C 0.000 }
gfCNCPoint4[28729] = {X 157.8634, Y 21.4565, Z -6.3333, A 0.000, B 0.000, C 0.000 }
gfCNCPoint4[28730] = {X 157.0798, Y 21.2109, Z -6.3333, A 0.000, B 0.000, C 0.000 }
gfCNCPoint4[28731] = {X 156.3606, Y 20.8144, Z -6.3333, A 0.000, B 0.000, C 0.000 }
gfCNCPoint4[28732] = {X 155.7346, Y 20.2829, Z -6.3333, A 0.000, B 0.000, C 0.000 }
gfCNCPoint4[28733] = {X 155.2267, Y 19.6375, Z -6.3333, A 0.000, B 0.000, C 0.000 }
gfCNCPoint4[28734] = {X 152.0370, Y 19.6387, Z -6.3333, A 0.000, B 0.000, C 0.000 }
gfCNCPoint4[28735] = {X 152.0358, Y 40.9684, Z -6.3333, A 0.000, B 0.000, C 0.000 }
gfCNCPoint4[28736] = {X 152.5609, Y 41.5338, Z -6.3333, A 0.000, B 0.000, C 0.000 }
gfCNCPoint4[28737] = {X 152.6512, Y 41.6413, Z -6.3333, A 0.000, B 0.000, C 0.000 }
gfCNCPoint4[28738] = {X 153.1470, Y 42.4207, Z -6.3333, A 0.000, B 0.000, C 0.000 }
gfCNCPoint4[28739] = {X 153.4562, Y 43.2911, Z -6.3333, A 0.000, B 0.000, C 0.000 }
gfCNCPoint4[28740] = {X 153.5631, Y 44.2086, Z -6.3333, A 0.000, B 0.000, C 0.000 }
gfCNCPoint4[28741] = {X 153.5629, Y 45.0392, Z -6.3333, A 0.000, B 0.000, C 0.000 }
gfCNCPoint4[28742] = {X 153.4532, Y 45.9406, Z -6.3333, A 0.000, B 0.000, C 0.000 }
gfCNCPoint4[28743] = {X 153.1468, Y 46.7954, Z -6.3333, A 0.000, B 0.000, C 0.000 }
gfCNCPoint4[28744] = {X 152.6589, Y 47.5613, Z -6.3333, A 0.000, B 0.000, C 0.000 }
gfCNCPoint4[28745] = {X 152.0138, Y 48.2003, Z -6.3333, A 0.000, B 0.000, C 0.000 }
gfCNCPoint4[28746] = {X 151.2432, Y 48.6808, Z -6.3333, A 0.000, B 0.000, C 0.000 }
gfCNCPoint4[28747] = {X 150.3855, Y 48.9789, Z -6.3333, A 0.000, B 0.000, C 0.000 }
gfCNCPoint4[28748] = {X 149.4831, Y 49.0800, Z -6.3333, A 0.000, B 0.000, C 0.000 }
gfCNCPoint4[28749] = {X 143.0396, Y 49.0800, Z -6.3333, A 0.000, B 0.000, C 0.000 }
gfCNCPoint4[28750] = {X 142.1362, Y 48.9787, Z -6.3333, A 0.000, B 0.000, C 0.000 }
gfCNCPoint4[28751] = {X 141.2777, Y 48.6799, Z -6.3333, A 0.000, B 0.000, C 0.000 }
gfCNCPoint4[28752] = {X 140.5066, Y 48.1985, Z -6.3333, A 0.000, B 0.000, C 0.000 }
gfCNCPoint4[28753] = {X 139.8613, Y 47.5582, Z -6.3333, A 0.000, B 0.000, C 0.000 }
gfCNCPoint4[28754] = {X 139.3737, Y 46.7910, Z -6.3333, A 0.000, B 0.000, C 0.000 }
gfCNCPoint4[28755] = {X 139.0682, Y 45.9349, Z -6.3333, A 0.000, B 0.000, C 0.000 }
gfCNCPoint4[28756] = {X 138.9598, Y 45.0323, Z -6.3333, A 0.000, B 0.000, C 0.000 }
gfCNCPoint4[28757] = {X 138.9600, Y 44.1527, Z -6.3333, A 0.000, B 0.000, C 0.000 }
gfCNCPoint4[28758] = {X 139.0706, Y 43.2637, Z -6.3333, A 0.000, B 0.000, C 0.000 }
gfCNCPoint4[28759] = {X 139.3725, Y 42.4203, Z -6.3333, A 0.000, B 0.000, C 0.000 }
gfCNCPoint4[28760] = {X 139.8512, Y 41.6631, Z -6.3333, A 0.000, B 0.000, C 0.000 }
gfCNCPoint4[28761] = {X 140.4836, Y 41.0287, Z -6.3333, A 0.000, B 0.000, C 0.000 }
gfCNCPoint4[28762] = {X 140.4836, Y 30.3968, Z -6.3333, A 0.000, B 0.000, C 0.000 }
gfCNCPoint4[28763] = {X 136.4836, Y 30.3968, Z -6.3333, A 0.000, B 0.000, C 0.000 }
gfCNCPoint4[28764] = {X 140.5636, Y 30.3968, Z -6.3333, A 0.000, B 0.000, C 0.000 }
gfCNCPoint4[28765] = {X 140.5636, Y 19.9580, Z -6.3333, A 0.000, B 0.000, C 0.000 }
gfCNCPoint4[28766] = {X 140.5638, Y 19.5580, Z -6.3333, A 0.000, B 0.000, C 0.000 }
gfCNCPoint4[28767] = {X 137.2663, Y 19.5575, Z -6.3333, A 0.000, B 0.000, C 0.000 }
gfCNCPoint4[28768] = {X 137.2444, Y 19.5615, Z -6.3333, A 0.000, B 0.000, C 0.000 }
gfCNCPoint4[28769] = {X 137.1364, Y 19.7307, Z -6.3333, A 0.000, B 0.000, C 0.000 }
gfCNCPoint4[28770] = {X 136.4969, Y 20.4537, Z -6.3333, A 0.000, B 0.000, C 0.000 }
gfCNCPoint4[28771] = {X 135.7028, Y 21.0025, Z -6.3333, A 0.000, B 0.000, C 0.000 }
gfCNCPoint4[28772] = {X 134.8004, Y 21.3451, Z -6.3333, A 0.000, B 0.000, C 0.000 }
gfCNCPoint4[28773] = {X 133.8422, Y 21.4615, Z -6.3333, A 0.000, B 0.000, C 0.000 }
gfCNCPoint4[28774] = {X 133.2006, Y 21.4615, Z -6.3333, A 0.000, B 0.000, C 0.000 }
gfCNCPoint4[28775] = {X 132.3106, Y 21.3612, Z -6.3333, A 0.000, B 0.000, C 0.000 }
gfCNCPoint4[28776] = {X 131.4651, Y 21.0654, Z -6.3333, A 0.000, B 0.000, C 0.000 }
gfCNCPoint4[28777] = {X 130.7067, Y 20.5889, Z -6.3333, A 0.000, B 0.000, C 0.000 }
gfCNCPoint4[28778] = {X 130.0733, Y 19.9555, Z -6.3333, A 0.000, B 0.000, C 0.000 }
gfCNCPoint4[28779] = {X 129.5968, Y 19.1971, Z -6.3333, A 0.000, B 0.000, C 0.000 }
gfCNCPoint4[28780] = {X 129.3009, Y 18.3516, Z -6.3333, A 0.000, B 0.000, C 0.000 }
gfCNCPoint4[28781] = {X 129.2006, Y 17.4615, Z -6.3333, A 0.000, B 0.000, C 0.000 }
gfCNCPoint4[28782] = {X 129.2006, Y 10.4835, Z -6.3333, A 0.000, B 0.000, C 0.000 }
gfCNCPoint4[28783] = {X 129.3009, Y 9.5934, Z -6.3333, A 0.000, B 0.000, C 0.000 }
gfCNCPoint4[28784] = {X 129.5968, Y 8.7480, Z -6.3333, A 0.000, B 0.000, C 0.000 }
gfCNCPoint4[28785] = {X 130.0733, Y 7.9896, Z -6.3333, A 0.000, B 0.000, C 0.000 }
gfCNCPoint4[28786] = {X 130.7067, Y 7.3562, Z -6.3333, A 0.000, B 0.000, C 0.000 }
gfCNCPoint4[28787] = {X 131.4651, Y 6.8796, Z -6.3333, A 0.000, B 0.000, C 0.000 }
gfCNCPoint4[28788] = {X 132.3106, Y 6.5838, Z -6.3333, A 0.000, B 0.000, C 0.000 }
